LIN {X 55.431,Y 89.332,Z 63.210,A 180.000,B 0.000,C 180.000} C_DIS
LIN {X 55.354,Y 89.351,Z 63.208,A 180.000,B 0.000,C 180.000} C_DIS
LIN {X 55.279,Y 89.372,Z 63.205,A 180.000,B 0.000,C 180.000} C_DIS
LIN {X 55.127,Y 89.416,Z 63.199,A 180.000,B 0.000,C 180.000} C_DIS
LIN {X 55.052,Y 89.438,Z 63.197,A 180.000,B 0.000,C 180.000} C_DIS
LIN {X 54.901,Y 89.482,Z 63.191,A 180.000,B 0.000,C 180.000} C_DIS
LIN {X 54.749,Y 89.526,Z 63.186,A 180.000,B 0.000,C 180.000} C_DIS
LIN {X 54.674,Y 89.548,Z 63.183,A 180.000,B 0.000,C 180.000} C_DIS
LIN {X 54.599,Y 89.572,Z 63.180,A 180.000,B 0.000,C 180.000} C_DIS
LIN {X 54.524,Y 89.598,Z 63.177,A 180.000,B 0.000,C 180.000} C_DIS
LIN {X 54.450,Y 89.625,Z 63.175,A 180.000,B 0.000,C 180.000} C_DIS
LIN {X 54.302,Y 89.678,Z 63.169,A 180.000,B 0.000,C 180.000} C_DIS
LIN {X 54.006,Y 89.785,Z 63.158,A 180.000,B 0.000,C 180.000} C_DIS
LIN {X 53.932,Y 89.812,Z 63.155,A 180.000,B 0.000,C 180.000} C_DIS
LIN {X 53.858,Y 89.840,Z 63.153,A 180.000,B 0.000,C 180.000} C_DIS
LIN {X 53.786,Y 89.871,Z 63.150,A 180.000,B 0.000,C 180.000} C_DIS
LIN {X 53.352,Y 90.058,Z 63.133,A 180.000,B 0.000,C 180.000} C_DIS
LIN {X 53.280,Y 90.090,Z 63.131,A 180.000,B 0.000,C 180.000} C_DIS
LIN {X 53.208,Y 90.121,Z 63.128,A 180.000,B 0.000,C 180.000} C_DIS
LIN {X 53.136,Y 90.154,Z 63.125,A 180.000,B 0.000,C 180.000} C_DIS
LIN {X 53.066,Y 90.189,Z 63.122,A 180.000,B 0.000,C 180.000} C_DIS
LIN {X 52.925,Y 90.261,Z 63.117,A 180.000,B 0.000,C 180.000} C_DIS
LIN {X 52.575,Y 90.440,Z 63.103,A 180.000,B 0.000,C 180.000} C_DIS
LIN {X 52.504,Y 90.475,Z 63.100,A 180.000,B 0.000,C 180.000} C_DIS
LIN {X 52.435,Y 90.513,Z 63.098,A 180.000,B 0.000,C 180.000} C_DIS
LIN {X 52.367,Y 90.552,Z 63.095,A 180.000,B 0.000,C 180.000} C_DIS
LIN {X 51.892,Y 90.833,Z 63.076,A 180.000,B 0.000,C 180.000} C_DIS
LIN {X 51.825,Y 90.873,Z 63.073,A 180.000,B 0.000,C 180.000} C_DIS
LIN {X 51.758,Y 90.915,Z 63.070,A 180.000,B 0.000,C 180.000} C_DIS
LIN {X 51.692,Y 90.959,Z 63.067,A 180.000,B 0.000,C 180.000} C_DIS
LIN {X 51.302,Y 91.224,Z 63.051,A 180.000,B 0.000,C 180.000} C_DIS
LIN {X 51.236,Y 91.268,Z 63.048,A 180.000,B 0.000,C 180.000} C_DIS
LIN {X 51.171,Y 91.313,Z 63.045,A 180.000,B 0.000,C 180.000} C_DIS
LIN {X 51.107,Y 91.359,Z 63.043,A 180.000,B 0.000,C 180.000} C_DIS
LIN {X 51.045,Y 91.406,Z 63.040,A 180.000,B 0.000,C 180.000} C_DIS
LIN {X 50.609,Y 91.744,Z 63.021,A 180.000,B 0.000,C 180.000} C_DIS
LIN {X 50.547,Y 91.792,Z 63.018,A 180.000,B 0.000,C 180.000} C_DIS
LIN {X 50.486,Y 91.842,Z 63.015,A 180.000,B 0.000,C 180.000} C_DIS
LIN {X 50.426,Y 91.894,Z 63.012,A 180.000,B 0.000,C 180.000} C_DIS
LIN {X 50.013,Y 92.258,Z 62.993,A 180.000,B 0.000,C 180.000} C_DIS
LIN {X 49.954,Y 92.310,Z 62.990,A 180.000,B 0.000,C 180.000} C_DIS
LIN {X 49.896,Y 92.364,Z 62.988,A 180.000,B 0.000,C 180.000} C_DIS
LIN {X 49.840,Y 92.419,Z 62.985,A 180.000,B 0.000,C 180.000} C_DIS
LIN {X 49.450,Y 92.809,Z 62.966,A 180.000,B 0.000,C 180.000} C_DIS
LIN {X 49.394,Y 92.865,Z 62.963,A 180.000,B 0.000,C 180.000} C_DIS
LIN {X 49.340,Y 92.921,Z 62.960,A 180.000,B 0.000,C 180.000} C_DIS
LIN {X 49.287,Y 92.980,Z 62.957,A 180.000,B 0.000,C 180.000} C_DIS
LIN {X 48.975,Y 93.334,Z 62.941,A 180.000,B 0.000,C 180.000} C_DIS
LIN {X 48.923,Y 93.393,Z 62.938,A 180.000,B 0.000,C 180.000} C_DIS
LIN {X 48.871,Y 93.453,Z 62.935,A 180.000,B 0.000,C 180.000} C_DIS
LIN {X 48.820,Y 93.513,Z 62.933,A 180.000,B 0.000,C 180.000} C_DIS
LIN {X 48.771,Y 93.575,Z 62.930,A 180.000,B 0.000,C 180.000} C_DIS
LIN {X 48.433,Y 94.010,Z 62.911,A 180.000,B 0.000,C 180.000} C_DIS
LIN {X 48.385,Y 94.072,Z 62.908,A 180.000,B 0.000,C 180.000} C_DIS
LIN {X 48.338,Y 94.136,Z 62.905,A 180.000,B 0.000,C 180.000} C_DIS
LIN {X 48.293,Y 94.200,Z 62.902,A 180.000,B 0.000,C 180.000} C_DIS
LIN {X 48.204,Y 94.331,Z 62.897,A 180.000,B 0.000,C 180.000} C_DIS
LIN {X 47.983,Y 94.656,Z 62.883,A 180.000,B 0.000,C 180.000} C_DIS
LIN {X 47.939,Y 94.721,Z 62.880,A 180.000,B 0.000,C 180.000} C_DIS
LIN {X 47.896,Y 94.788,Z 62.878,A 180.000,B 0.000,C 180.000} C_DIS
LIN {X 47.855,Y 94.855,Z 62.875,A 180.000,B 0.000,C 180.000} C_DIS
LIN {X 47.615,Y 95.262,Z 62.858,A 180.000,B 0.000,C 180.000} C_DIS
LIN {X 47.575,Y 95.329,Z 62.856,A 180.000,B 0.000,C 180.000} C_DIS
LIN {X 47.535,Y 95.397,Z 62.853,A 180.000,B 0.000,C 180.000} C_DIS
LIN {X 47.496,Y 95.466,Z 62.850,A 180.000,B 0.000,C 180.000} C_DIS
LIN {X 47.459,Y 95.536,Z 62.847,A 180.000,B 0.000,C 180.000} C_DIS
LIN {X 47.388,Y 95.676,Z 62.842,A 180.000,B 0.000,C 180.000} C_DIS
LIN {X 47.209,Y 96.027,Z 62.828,A 180.000,B 0.000,C 180.000} C_DIS
LIN {X 47.173,Y 96.097,Z 62.825,A 180.000,B 0.000,C 180.000} C_DIS
LIN {X 47.139,Y 96.168,Z 62.823,A 180.000,B 0.000,C 180.000} C_DIS
LIN {X 47.107,Y 96.240,Z 62.820,A 180.000,B 0.000,C 180.000} C_DIS
LIN {X 47.044,Y 96.384,Z 62.814,A 180.000,B 0.000,C 180.000} C_DIS
LIN {X 47.013,Y 96.457,Z 62.812,A 180.000,B 0.000,C 180.000} C_DIS
LIN {X 46.951,Y 96.601,Z 62.806,A 180.000,B 0.000,C 180.000} C_DIS
LIN {X 46.888,Y 96.746,Z 62.801,A 180.000,B 0.000,C 180.000} C_DIS
LIN {X 46.857,Y 96.818,Z 62.798,A 180.000,B 0.000,C 180.000} C_DIS
LIN {X 46.827,Y 96.891,Z 62.795,A 180.000,B 0.000,C 180.000} C_DIS
LIN {X 46.800,Y 96.965,Z 62.792,A 180.000,B 0.000,C 180.000} C_DIS
LIN {X 46.773,Y 97.039,Z 62.790,A 180.000,B 0.000,C 180.000} C_DIS
LIN {X 46.720,Y 97.187,Z 62.784,A 180.000,B 0.000,C 180.000} C_DIS
LIN {X 46.639,Y 97.409,Z 62.776,A 180.000,B 0.000,C 180.000} C_DIS
LIN {X 46.613,Y 97.483,Z 62.773,A 180.000,B 0.000,C 180.000} C_DIS
LIN {X 46.586,Y 97.557,Z 62.770,A 180.000,B 0.000,C 180.000} C_DIS
LIN {X 46.561,Y 97.632,Z 62.768,A 180.000,B 0.000,C 180.000} C_DIS
LIN {X 46.538,Y 97.707,Z 62.765,A 180.000,B 0.000,C 180.000} C_DIS
LIN {X 46.494,Y 97.859,Z 62.759,A 180.000,B 0.000,C 180.000} C_DIS
LIN {X 46.472,Y 97.934,Z 62.757,A 180.000,B 0.000,C 180.000} C_DIS
LIN {X 46.428,Y 98.085,Z 62.751,A 180.000,B 0.000,C 180.000} C_DIS
LIN {X 46.384,Y 98.237,Z 62.746,A 180.000,B 0.000,C 180.000} C_DIS
LIN {X 46.362,Y 98.312,Z 62.743,A 180.000,B 0.000,C 180.000} C_DIS
LIN {X 46.342,Y 98.388,Z 62.740,A 180.000,B 0.000,C 180.000} C_DIS
LIN {X 46.324,Y 98.465,Z 62.737,A 180.000,B 0.000,C 180.000} C_DIS
LIN {X 46.307,Y 98.542,Z 62.735,A 180.000,B 0.000,C 180.000} C_DIS
LIN {X 46.272,Y 98.696,Z 62.729,A 180.000,B 0.000,C 180.000} C_DIS
LIN {X 46.221,Y 98.926,Z 62.721,A 180.000,B 0.000,C 180.000} C_DIS
LIN {X 46.204,Y 99.003,Z 62.718,A 180.000,B 0.000,C 180.000} C_DIS
LIN {X 46.186,Y 99.080,Z 62.715,A 180.000,B 0.000,C 180.000} C_DIS
LIN {X 46.171,Y 99.157,Z 62.713,A 180.000,B 0.000,C 180.000} C_DIS
LIN {X 46.157,Y 99.235,Z 62.710,A 180.000,B 0.000,C 180.000} C_DIS
LIN {X 46.133,Y 99.390,Z 62.704,A 180.000,B 0.000,C 180.000} C_DIS
LIN {X 46.120,Y 99.468,Z 62.702,A 180.000,B 0.000,C 180.000} C_DIS
LIN {X 46.096,Y 99.624,Z 62.696,A 180.000,B 0.000,C 180.000} C_DIS
LIN {X 46.071,Y 99.779,Z 62.691,A 180.000,B 0.000,C 180.000} C_DIS
LIN {X 46.059,Y 99.857,Z 62.688,A 180.000,B 0.000,C 180.000} C_DIS
LIN {X 46.048,Y 99.935,Z 62.685,A 180.000,B 0.000,C 180.000} C_DIS
LIN {X 46.040,Y 100.013,Z 62.682,A 180.000,B 0.000,C 180.000} C_DIS
LIN {X 46.025,Y 100.170,Z 62.677,A 180.000,B 0.000,C 180.000} C_DIS
LIN {X 46.010,Y 100.327,Z 62.672,A 180.000,B 0.000,C 180.000} C_DIS
LIN {X 45.995,Y 100.484,Z 62.666,A 180.000,B 0.000,C 180.000} C_DIS
LIN {X 45.988,Y 100.562,Z 62.664,A 180.000,B 0.000,C 180.000} C_DIS
LIN {X 45.980,Y 100.640,Z 62.661,A 180.000,B 0.000,C 180.000} C_DIS
LIN {X 45.974,Y 100.719,Z 62.659,A 180.000,B 0.000,C 180.000} C_DIS
LIN {X 45.971,Y 100.798,Z 62.656,A 180.000,B 0.000,C 180.000} C_DIS
LIN {X 45.968,Y 100.876,Z 62.654,A 180.000,B 0.000,C 180.000} C_DIS
LIN {X 45.966,Y 100.955,Z 62.651,A 180.000,B 0.000,C 180.000} C_DIS
LIN {X 45.963,Y 101.034,Z 62.649,A 180.000,B 0.000,C 180.000} C_DIS
LIN {X 45.958,Y 101.191,Z 62.644,A 180.000,B 0.000,C 180.000} C_DIS
LIN {X 45.954,Y 101.349,Z 62.639,A 180.000,B 0.000,C 180.000} C_DIS
LIN {X 45.950,Y 101.506,Z 62.634,A 180.000,B 0.000,C 180.000} C_DIS
LIN {X 45.954,Y 101.664,Z 62.629,A 180.000,B 0.000,C 180.000} C_DIS
LIN {X 45.959,Y 101.821,Z 62.624,A 180.000,B 0.000,C 180.000} C_DIS
LIN {X 45.964,Y 101.978,Z 62.620,A 180.000,B 0.000,C 180.000} C_DIS
LIN {X 45.969,Y 102.136,Z 62.615,A 180.000,B 0.000,C 180.000} C_DIS
LIN {X 45.975,Y 102.293,Z 62.611,A 180.000,B 0.000,C 180.000} C_DIS
LIN {X 45.989,Y 102.450,Z 62.606,A 180.000,B 0.000,C 180.000} C_DIS
LIN {X 46.004,Y 102.607,Z 62.602,A 180.000,B 0.000,C 180.000} C_DIS
LIN {X 46.018,Y 102.764,Z 62.597,A 180.000,B 0.000,C 180.000} C_DIS
LIN {X 46.033,Y 102.920,Z 62.593,A 180.000,B 0.000,C 180.000} C_DIS
LIN {X 46.049,Y 103.077,Z 62.589,A 180.000,B 0.000,C 180.000} C_DIS
LIN {X 46.073,Y 103.233,Z 62.585,A 180.000,B 0.000,C 180.000} C_DIS
LIN {X 46.098,Y 103.388,Z 62.581,A 180.000,B 0.000,C 180.000} C_DIS
LIN {X 46.122,Y 103.544,Z 62.577,A 180.000,B 0.000,C 180.000} C_DIS
LIN {X 46.147,Y 103.700,Z 62.573,A 180.000,B 0.000,C 180.000} C_DIS
LIN {X 46.173,Y 103.855,Z 62.570,A 180.000,B 0.000,C 180.000} C_DIS
LIN {X 46.206,Y 104.009,Z 62.566,A 180.000,B 0.000,C 180.000} C_DIS
LIN {X 46.241,Y 104.163,Z 62.562,A 180.000,B 0.000,C 180.000} C_DIS
LIN {X 46.275,Y 104.316,Z 62.559,A 180.000,B 0.000,C 180.000} C_DIS
LIN {X 46.309,Y 104.470,Z 62.556,A 180.000,B 0.000,C 180.000} C_DIS
LIN {X 46.345,Y 104.623,Z 62.552,A 180.000,B 0.000,C 180.000} C_DIS
LIN {X 46.388,Y 104.775,Z 62.549,A 180.000,B 0.000,C 180.000} C_DIS
LIN {X 46.432,Y 104.926,Z 62.546,A 180.000,B 0.000,C 180.000} C_DIS
LIN {X 46.476,Y 105.077,Z 62.543,A 180.000,B 0.000,C 180.000} C_DIS
LIN {X 46.520,Y 105.229,Z 62.540,A 180.000,B 0.000,C 180.000} C_DIS
LIN {X 46.565,Y 105.380,Z 62.537,A 180.000,B 0.000,C 180.000} C_DIS
LIN {X 46.617,Y 105.528,Z 62.534,A 180.000,B 0.000,C 180.000} C_DIS
LIN {X 46.670,Y 105.676,Z 62.532,A 180.000,B 0.000,C 180.000} C_DIS
LIN {X 46.724,Y 105.825,Z 62.529,A 180.000,B 0.000,C 180.000} C_DIS
LIN {X 46.777,Y 105.973,Z 62.527,A 180.000,B 0.000,C 180.000} C_DIS
LIN {X 46.893,Y 106.266,Z 62.522,A 180.000,B 0.000,C 180.000} C_DIS
LIN {X 47.018,Y 106.555,Z 62.518,A 180.000,B 0.000,C 180.000} C_DIS
LIN {X 47.144,Y 106.843,Z 62.514,A 180.000,B 0.000,C 180.000} C_DIS
LIN {X 47.286,Y 107.125,Z 62.511,A 180.000,B 0.000,C 180.000} C_DIS
LIN {X 47.429,Y 107.405,Z 62.508,A 180.000,B 0.000,C 180.000} C_DIS
LIN {X 47.581,Y 107.681,Z 62.505,A 180.000,B 0.000,C 180.000} C_DIS
LIN {X 47.741,Y 107.952,Z 62.503,A 180.000,B 0.000,C 180.000} C_DIS
LIN {X 47.903,Y 108.223,Z 62.502,A 180.000,B 0.000,C 180.000} C_DIS
LIN {X 48.079,Y 108.484,Z 62.501,A 180.000,B 0.000,C 180.000} C_DIS
LIN {X 48.256,Y 108.745,Z 62.500,A 180.000,B 0.000,C 180.000} C_DIS
LIN {X 48.390,Y 108.933,Z 62.500,A 180.000,B 0.000,C 180.000} C_DIS
; Cutting Move Starts
LIN {X 48.450,Y 109.012,Z 62.500,A 180.000,B 0.000,C 180.000} C_DIS
LIN {X 48.759,Y 109.410,Z 62.500,A 180.000,B 0.000,C 180.000} C_DIS
LIN {X 48.807,Y 109.472,Z 62.500,A 180.000,B 0.000,C 180.000} C_DIS
LIN {X 48.907,Y 109.589,Z 62.500,A 180.000,B 0.000,C 180.000} C_DIS
LIN {X 49.223,Y 109.947,Z 62.500,A 180.000,B 0.000,C 180.000} C_DIS
LIN {X 49.344,Y 110.083,Z 62.500,A 180.000,B 0.000,C 180.000} C_DIS
LIN {X 49.384,Y 110.126,Z 62.500,A 180.000,B 0.000,C 180.000} C_DIS
LIN {X 49.523,Y 110.264,Z 62.500,A 180.000,B 0.000,C 180.000} C_DIS
LIN {X 49.742,Y 110.483,Z 62.500,A 180.000,B 0.000,C 180.000} C_DIS
LIN {X 49.880,Y 110.621,Z 62.500,A 180.000,B 0.000,C 180.000} C_DIS
LIN {X 49.923,Y 110.662,Z 62.500,A 180.000,B 0.000,C 180.000} C_DIS
LIN {X 50.059,Y 110.782,Z 62.500,A 180.000,B 0.000,C 180.000} C_DIS
LIN {X 50.416,Y 111.098,Z 62.500,A 180.000,B 0.000,C 180.000} C_DIS
LIN {X 50.535,Y 111.198,Z 62.500,A 180.000,B 0.000,C 180.000} C_DIS
LIN {X 50.595,Y 111.245,Z 62.500,A 180.000,B 0.000,C 180.000} C_DIS
LIN {X 50.996,Y 111.556,Z 62.500,A 180.000,B 0.000,C 180.000} C_DIS
LIN {X 51.131,Y 111.659,Z 62.500,A 180.000,B 0.000,C 180.000} C_DIS
LIN {X 51.241,Y 111.734,Z 62.500,A 180.000,B 0.000,C 180.000} C_DIS
LIN {X 51.668,Y 112.025,Z 62.500,A 180.000,B 0.000,C 180.000} C_DIS
LIN {X 51.769,Y 112.092,Z 62.500,A 180.000,B 0.000,C 180.000} C_DIS
LIN {X 51.847,Y 112.140,Z 62.500,A 180.000,B 0.000,C 180.000} C_DIS
LIN {X 52.383,Y 112.457,Z 62.500,A 180.000,B 0.000,C 180.000} C_DIS
LIN {X 52.562,Y 112.554,Z 62.500,A 180.000,B 0.000,C 180.000} C_DIS
LIN {X 53.059,Y 112.807,Z 62.500,A 180.000,B 0.000,C 180.000} C_DIS
LIN {X 53.098,Y 112.827,Z 62.500,A 180.000,B 0.000,C 180.000} C_DIS
LIN {X 53.277,Y 112.909,Z 62.500,A 180.000,B 0.000,C 180.000} C_DIS
LIN {X 53.813,Y 113.141,Z 62.500,A 180.000,B 0.000,C 180.000} C_DIS
LIN {X 53.870,Y 113.165,Z 62.500,A 180.000,B 0.000,C 180.000} C_DIS
LIN {X 53.992,Y 113.210,Z 62.500,A 180.000,B 0.000,C 180.000} C_DIS
LIN {X 54.528,Y 113.403,Z 62.500,A 180.000,B 0.000,C 180.000} C_DIS
LIN {X 54.707,Y 113.462,Z 62.500,A 180.000,B 0.000,C 180.000} C_DIS
LIN {X 55.243,Y 113.618,Z 62.500,A 180.000,B 0.000,C 180.000} C_DIS
LIN {X 55.422,Y 113.666,Z 62.500,A 180.000,B 0.000,C 180.000} C_DIS
LIN {X 55.575,Y 113.701,Z 62.500,A 180.000,B 0.000,C 180.000} C_DIS
LIN {X 55.958,Y 113.786,Z 62.500,A 180.000,B 0.000,C 180.000} C_DIS
LIN {X 56.137,Y 113.826,Z 62.500,A 180.000,B 0.000,C 180.000} C_DIS
LIN {X 56.316,Y 113.855,Z 62.500,A 180.000,B 0.000,C 180.000} C_DIS
LIN {X 56.852,Y 113.940,Z 62.500,A 180.000,B 0.000,C 180.000} C_DIS
LIN {X 57.031,Y 113.962,Z 62.500,A 180.000,B 0.000,C 180.000} C_DIS
LIN {X 57.567,Y 114.013,Z 62.500,A 180.000,B 0.000,C 180.000} C_DIS
LIN {X 57.746,Y 114.027,Z 62.500,A 180.000,B 0.000,C 180.000} C_DIS
LIN {X 57.925,Y 114.033,Z 62.500,A 180.000,B 0.000,C 180.000} C_DIS
LIN {X 58.282,Y 114.044,Z 62.500,A 180.000,B 0.000,C 180.000} C_DIS
LIN {X 58.461,Y 114.050,Z 62.500,A 180.000,B 0.000,C 180.000} C_DIS
LIN {X 58.640,Y 114.047,Z 62.500,A 180.000,B 0.000,C 180.000} C_DIS
LIN {X 59.176,Y 114.030,Z 62.500,A 180.000,B 0.000,C 180.000} C_DIS
LIN {X 59.355,Y 114.020,Z 62.500,A 180.000,B 0.000,C 180.000} C_DIS
LIN {X 59.534,Y 114.003,Z 62.500,A 180.000,B 0.000,C 180.000} C_DIS
LIN {X 59.891,Y 113.969,Z 62.500,A 180.000,B 0.000,C 180.000} C_DIS
LIN {X 60.070,Y 113.951,Z 62.500,A 180.000,B 0.000,C 180.000} C_DIS
LIN {X 60.249,Y 113.924,Z 62.500,A 180.000,B 0.000,C 180.000} C_DIS
LIN {X 60.606,Y 113.868,Z 62.500,A 180.000,B 0.000,C 180.000} C_DIS
LIN {X 60.785,Y 113.839,Z 62.500,A 180.000,B 0.000,C 180.000} C_DIS
LIN {X 60.964,Y 113.804,Z 62.500,A 180.000,B 0.000,C 180.000} C_DIS
LIN {X 61.500,Y 113.684,Z 62.500,A 180.000,B 0.000,C 180.000} C_DIS
LIN {X 61.679,Y 113.640,Z 62.500,A 180.000,B 0.000,C 180.000} C_DIS
LIN {X 61.858,Y 113.588,Z 62.500,A 180.000,B 0.000,C 180.000} C_DIS
LIN {X 62.215,Y 113.484,Z 62.500,A 180.000,B 0.000,C 180.000} C_DIS
LIN {X 62.394,Y 113.431,Z 62.500,A 180.000,B 0.000,C 180.000} C_DIS
LIN {X 62.573,Y 113.367,Z 62.500,A 180.000,B 0.000,C 180.000} C_DIS
LIN {X 62.930,Y 113.238,Z 62.500,A 180.000,B 0.000,C 180.000} C_DIS
LIN {X 63.109,Y 113.173,Z 62.500,A 180.000,B 0.000,C 180.000} C_DIS
LIN {X 63.130,Y 113.165,Z 62.500,A 180.000,B 0.000,C 180.000} C_DIS
LIN {X 63.288,Y 113.097,Z 62.500,A 180.000,B 0.000,C 180.000} C_DIS
LIN {X 63.645,Y 112.943,Z 62.500,A 180.000,B 0.000,C 180.000} C_DIS
LIN {X 63.824,Y 112.865,Z 62.500,A 180.000,B 0.000,C 180.000} C_DIS
LIN {X 63.941,Y 112.807,Z 62.500,A 180.000,B 0.000,C 180.000} C_DIS
LIN {X 64.360,Y 112.594,Z 62.500,A 180.000,B 0.000,C 180.000} C_DIS
LIN {X 64.539,Y 112.501,Z 62.500,A 180.000,B 0.000,C 180.000} C_DIS
LIN {X 64.630,Y 112.450,Z 62.500,A 180.000,B 0.000,C 180.000} C_DIS
LIN {X 65.075,Y 112.186,Z 62.500,A 180.000,B 0.000,C 180.000} C_DIS
LIN {X 65.231,Y 112.092,Z 62.500,A 180.000,B 0.000,C 180.000} C_DIS
LIN {X 65.254,Y 112.077,Z 62.500,A 180.000,B 0.000,C 180.000} C_DIS
LIN {X 65.433,Y 111.956,Z 62.500,A 180.000,B 0.000,C 180.000} C_DIS
LIN {X 65.791,Y 111.713,Z 62.500,A 180.000,B 0.000,C 180.000} C_DIS
LIN {X 65.969,Y 111.583,Z 62.500,A 180.000,B 0.000,C 180.000} C_DIS
LIN {X 66.327,Y 111.306,Z 62.500,A 180.000,B 0.000,C 180.000} C_DIS
LIN {X 66.465,Y 111.198,Z 62.500,A 180.000,B 0.000,C 180.000} C_DIS
LIN {X 66.506,Y 111.165,Z 62.500,A 180.000,B 0.000,C 180.000} C_DIS
LIN {X 66.672,Y 111.019,Z 62.500,A 180.000,B 0.000,C 180.000} C_DIS
LIN {X 66.875,Y 110.841,Z 62.500,A 180.000,B 0.000,C 180.000} C_DIS
LIN {X 67.042,Y 110.693,Z 62.500,A 180.000,B 0.000,C 180.000} C_DIS
LIN {X 67.077,Y 110.662,Z 62.500,A 180.000,B 0.000,C 180.000} C_DIS
LIN {X 67.221,Y 110.521,Z 62.500,A 180.000,B 0.000,C 180.000} C_DIS
LIN {X 67.578,Y 110.163,Z 62.500,A 180.000,B 0.000,C 180.000} C_DIS
LIN {X 67.616,Y 110.126,Z 62.500,A 180.000,B 0.000,C 180.000} C_DIS
LIN {X 67.757,Y 109.970,Z 62.500,A 180.000,B 0.000,C 180.000} C_DIS
LIN {X 68.115,Y 109.564,Z 62.500,A 180.000,B 0.000,C 180.000} C_DIS
LIN {X 68.241,Y 109.410,Z 62.500,A 180.000,B 0.000,C 180.000} C_DIS
LIN {X 68.518,Y 109.053,Z 62.500,A 180.000,B 0.000,C 180.000} C_DIS
LIN {X 68.651,Y 108.880,Z 62.500,A 180.000,B 0.000,C 180.000} C_DIS
LIN {X 68.655,Y 108.874,Z 62.500,A 180.000,B 0.000,C 180.000} C_DIS
LIN {X 68.778,Y 108.695,Z 62.500,A 180.000,B 0.000,C 180.000} C_DIS
LIN {X 69.021,Y 108.338,Z 62.500,A 180.000,B 0.000,C 180.000} C_DIS
LIN {X 69.137,Y 108.159,Z 62.500,A 180.000,B 0.000,C 180.000} C_DIS
LIN {X 69.454,Y 107.623,Z 62.500,A 180.000,B 0.000,C 180.000} C_DIS
LIN {X 69.545,Y 107.456,Z 62.500,A 180.000,B 0.000,C 180.000} C_DIS
LIN {X 69.733,Y 107.086,Z 62.500,A 180.000,B 0.000,C 180.000} C_DIS
LIN {X 69.824,Y 106.908,Z 62.500,A 180.000,B 0.000,C 180.000} C_DIS
LIN {X 69.902,Y 106.739,Z 62.500,A 180.000,B 0.000,C 180.000} C_DIS
LIN {X 70.139,Y 106.193,Z 62.500,A 180.000,B 0.000,C 180.000} C_DIS
LIN {X 70.208,Y 106.014,Z 62.500,A 180.000,B 0.000,C 180.000} C_DIS
LIN {X 70.401,Y 105.477,Z 62.500,A 180.000,B 0.000,C 180.000} C_DIS
LIN {X 70.439,Y 105.369,Z 62.500,A 180.000,B 0.000,C 180.000} C_DIS
LIN {X 70.460,Y 105.299,Z 62.500,A 180.000,B 0.000,C 180.000} C_DIS
LIN {X 70.617,Y 104.758,Z 62.500,A 180.000,B 0.000,C 180.000} C_DIS
LIN {X 70.665,Y 104.584,Z 62.500,A 180.000,B 0.000,C 180.000} C_DIS
LIN {X 70.705,Y 104.405,Z 62.500,A 180.000,B 0.000,C 180.000} C_DIS
LIN {X 70.796,Y 103.999,Z 62.500,A 180.000,B 0.000,C 180.000} C_DIS
LIN {X 70.824,Y 103.869,Z 62.500,A 180.000,B 0.000,C 180.000} C_DIS
LIN {X 70.855,Y 103.690,Z 62.500,A 180.000,B 0.000,C 180.000} C_DIS
LIN {X 70.940,Y 103.153,Z 62.500,A 180.000,B 0.000,C 180.000} C_DIS
LIN {X 70.962,Y 102.975,Z 62.500,A 180.000,B 0.000,C 180.000} C_DIS
LIN {X 71.012,Y 102.438,Z 62.500,A 180.000,B 0.000,C 180.000} C_DIS
LIN {X 71.027,Y 102.260,Z 62.500,A 180.000,B 0.000,C 180.000} C_DIS
LIN {X 71.033,Y 102.081,Z 62.500,A 180.000,B 0.000,C 180.000} C_DIS
LIN {X 71.044,Y 101.723,Z 62.500,A 180.000,B 0.000,C 180.000} C_DIS
LIN {X 71.050,Y 101.545,Z 62.500,A 180.000,B 0.000,C 180.000} C_DIS
LIN {X 71.047,Y 101.366,Z 62.500,A 180.000,B 0.000,C 180.000} C_DIS
LIN {X 71.030,Y 100.829,Z 62.500,A 180.000,B 0.000,C 180.000} C_DIS
LIN {X 71.021,Y 100.651,Z 62.500,A 180.000,B 0.000,C 180.000} C_DIS
LIN {X 71.004,Y 100.472,Z 62.500,A 180.000,B 0.000,C 180.000} C_DIS
LIN {X 70.970,Y 100.114,Z 62.500,A 180.000,B 0.000,C 180.000} C_DIS
LIN {X 70.952,Y 99.936,Z 62.500,A 180.000,B 0.000,C 180.000} C_DIS
LIN {X 70.925,Y 99.757,Z 62.500,A 180.000,B 0.000,C 180.000} C_DIS
LIN {X 70.840,Y 99.221,Z 62.500,A 180.000,B 0.000,C 180.000} C_DIS
LIN {X 70.805,Y 99.042,Z 62.500,A 180.000,B 0.000,C 180.000} C_DIS
LIN {X 70.718,Y 98.654,Z 62.500,A 180.000,B 0.000,C 180.000} C_DIS
LIN {X 70.685,Y 98.505,Z 62.500,A 180.000,B 0.000,C 180.000} C_DIS
LIN {X 70.642,Y 98.327,Z 62.500,A 180.000,B 0.000,C 180.000} C_DIS
LIN {X 70.617,Y 98.242,Z 62.500,A 180.000,B 0.000,C 180.000} C_DIS
LIN {X 70.486,Y 97.790,Z 62.500,A 180.000,B 0.000,C 180.000} C_DIS
LIN {X 70.439,Y 97.631,Z 62.500,A 180.000,B 0.000,C 180.000} C_DIS
LIN {X 70.432,Y 97.612,Z 62.500,A 180.000,B 0.000,C 180.000} C_DIS
LIN {X 70.369,Y 97.433,Z 62.500,A 180.000,B 0.000,C 180.000} C_DIS
LIN {X 70.240,Y 97.075,Z 62.500,A 180.000,B 0.000,C 180.000} C_DIS
LIN {X 70.175,Y 96.897,Z 62.500,A 180.000,B 0.000,C 180.000} C_DIS
LIN {X 70.100,Y 96.718,Z 62.500,A 180.000,B 0.000,C 180.000} C_DIS
LIN {X 69.902,Y 96.261,Z 62.500,A 180.000,B 0.000,C 180.000} C_DIS
LIN {X 69.867,Y 96.181,Z 62.500,A 180.000,B 0.000,C 180.000} C_DIS
LIN {X 69.779,Y 96.003,Z 62.500,A 180.000,B 0.000,C 180.000} C_DIS
LIN {X 69.545,Y 95.544,Z 62.500,A 180.000,B 0.000,C 180.000} C_DIS
LIN {X 69.504,Y 95.466,Z 62.500,A 180.000,B 0.000,C 180.000} C_DIS
LIN {X 69.401,Y 95.288,Z 62.500,A 180.000,B 0.000,C 180.000} C_DIS
LIN {X 69.187,Y 94.927,Z 62.500,A 180.000,B 0.000,C 180.000} C_DIS
LIN {X 69.081,Y 94.751,Z 62.500,A 180.000,B 0.000,C 180.000} C_DIS
LIN {X 69.008,Y 94.644,Z 62.500,A 180.000,B 0.000,C 180.000} C_DIS
LIN {X 68.717,Y 94.215,Z 62.500,A 180.000,B 0.000,C 180.000} C_DIS
LIN {X 68.651,Y 94.120,Z 62.500,A 180.000,B 0.000,C 180.000} C_DIS
LIN {X 68.587,Y 94.036,Z 62.500,A 180.000,B 0.000,C 180.000} C_DIS
LIN {X 68.293,Y 93.657,Z 62.500,A 180.000,B 0.000,C 180.000} C_DIS
LIN {X 68.170,Y 93.500,Z 62.500,A 180.000,B 0.000,C 180.000} C_DIS
LIN {X 68.115,Y 93.436,Z 62.500,A 180.000,B 0.000,C 180.000} C_DIS
LIN {X 67.698,Y 92.964,Z 62.500,A 180.000,B 0.000,C 180.000} C_DIS
LIN {X 67.578,Y 92.837,Z 62.500,A 180.000,B 0.000,C 180.000} C_DIS
LIN {X 67.169,Y 92.427,Z 62.500,A 180.000,B 0.000,C 180.000} C_DIS
LIN {X 67.061,Y 92.325,Z 62.500,A 180.000,B 0.000,C 180.000} C_DIS
LIN {X 67.042,Y 92.307,Z 62.500,A 180.000,B 0.000,C 180.000} C_DIS
LIN {X 66.976,Y 92.249,Z 62.500,A 180.000,B 0.000,C 180.000} C_DIS
LIN {X 66.571,Y 91.891,Z 62.500,A 180.000,B 0.000,C 180.000} C_DIS
LIN {X 66.506,Y 91.835,Z 62.500,A 180.000,B 0.000,C 180.000} C_DIS
LIN {X 66.350,Y 91.712,Z 62.500,A 180.000,B 0.000,C 180.000} C_DIS
LIN {X 65.969,Y 91.417,Z 62.500,A 180.000,B 0.000,C 180.000} C_DIS
LIN {X 65.887,Y 91.355,Z 62.500,A 180.000,B 0.000,C 180.000} C_DIS
LIN {X 65.791,Y 91.287,Z 62.500,A 180.000,B 0.000,C 180.000} C_DIS
LIN {X 65.364,Y 90.997,Z 62.500,A 180.000,B 0.000,C 180.000} C_DIS
LIN {X 65.254,Y 90.923,Z 62.500,A 180.000,B 0.000,C 180.000} C_DIS
LIN {X 65.083,Y 90.818,Z 62.500,A 180.000,B 0.000,C 180.000} C_DIS
LIN {X 64.718,Y 90.603,Z 62.500,A 180.000,B 0.000,C 180.000} C_DIS
LIN {X 64.539,Y 90.499,Z 62.500,A 180.000,B 0.000,C 180.000} C_DIS
LIN {X 64.467,Y 90.461,Z 62.500,A 180.000,B 0.000,C 180.000} C_DIS
LIN {X 64.003,Y 90.224,Z 62.500,A 180.000,B 0.000,C 180.000} C_DIS
LIN {X 63.824,Y 90.135,Z 62.500,A 180.000,B 0.000,C 180.000} C_DIS
LIN {X 63.752,Y 90.103,Z 62.500,A 180.000,B 0.000,C 180.000} C_DIS
LIN {X 63.288,Y 89.903,Z 62.500,A 180.000,B 0.000,C 180.000} C_DIS
LIN {X 63.109,Y 89.827,Z 62.500,A 180.000,B 0.000,C 180.000} C_DIS
LIN {X 62.930,Y 89.762,Z 62.500,A 180.000,B 0.000,C 180.000} C_DIS
LIN {X 62.573,Y 89.633,Z 62.500,A 180.000,B 0.000,C 180.000} C_DIS
LIN {X 62.394,Y 89.569,Z 62.500,A 180.000,B 0.000,C 180.000} C_DIS
LIN {X 62.387,Y 89.567,Z 62.500,A 180.000,B 0.000,C 180.000} C_DIS
LIN {X 62.215,Y 89.516,Z 62.500,A 180.000,B 0.000,C 180.000} C_DIS
LIN {X 61.777,Y 89.388,Z 62.500,A 180.000,B 0.000,C 180.000} C_DIS
LIN {X 61.679,Y 89.360,Z 62.500,A 180.000,B 0.000,C 180.000} C_DIS
LIN {X 61.500,Y 89.316,Z 62.500,A 180.000,B 0.000,C 180.000} C_DIS
LIN {X 60.964,Y 89.196,Z 62.500,A 180.000,B 0.000,C 180.000} C_DIS
LIN {X 60.785,Y 89.161,Z 62.500,A 180.000,B 0.000,C 180.000} C_DIS
LIN {X 60.606,Y 89.132,Z 62.500,A 180.000,B 0.000,C 180.000} C_DIS
LIN {X 60.249,Y 89.076,Z 62.500,A 180.000,B 0.000,C 180.000} C_DIS
LIN {X 60.070,Y 89.049,Z 62.500,A 180.000,B 0.000,C 180.000} C_DIS
LIN {X 59.892,Y 89.031,Z 62.500,A 180.000,B 0.000,C 180.000} C_DIS
LIN {X 59.534,Y 88.997,Z 62.500,A 180.000,B 0.000,C 180.000} C_DIS
LIN {X 59.355,Y 88.980,Z 62.500,A 180.000,B 0.000,C 180.000} C_DIS
LIN {X 59.176,Y 88.970,Z 62.500,A 180.000,B 0.000,C 180.000} C_DIS
LIN {X 58.640,Y 88.953,Z 62.500,A 180.000,B 0.000,C 180.000} C_DIS
LIN {X 58.461,Y 88.950,Z 62.500,A 180.000,B 0.000,C 180.000} C_DIS
LIN {X 58.282,Y 88.956,Z 62.500,A 180.000,B 0.000,C 180.000} C_DIS
LIN {X 57.925,Y 88.967,Z 62.500,A 180.000,B 0.000,C 180.000} C_DIS
LIN {X 57.746,Y 88.973,Z 62.500,A 180.000,B 0.000,C 180.000} C_DIS
LIN {X 57.567,Y 88.987,Z 62.500,A 180.000,B 0.000,C 180.000} C_DIS
LIN {X 57.031,Y 89.038,Z 62.500,A 180.000,B 0.000,C 180.000} C_DIS
LIN {X 56.852,Y 89.060,Z 62.500,A 180.000,B 0.000,C 180.000} C_DIS
LIN {X 56.316,Y 89.145,Z 62.500,A 180.000,B 0.000,C 180.000} C_DIS
LIN {X 56.137,Y 89.174,Z 62.500,A 180.000,B 0.000,C 180.000} C_DIS
LIN {X 55.977,Y 89.209,Z 62.500,A 180.000,B 0.000,C 180.000} C_DIS
LIN {X 55.601,Y 89.293,Z 62.500,A 180.000,B 0.000,C 180.000} C_DIS
LIN {X 55.422,Y 89.334,Z 62.500,A 180.000,B 0.000,C 180.000} C_DIS
LIN {X 55.243,Y 89.382,Z 62.500,A 180.000,B 0.000,C 180.000} C_DIS
LIN {X 54.707,Y 89.538,Z 62.500,A 180.000,B 0.000,C 180.000} C_DIS
LIN {X 54.613,Y 89.567,Z 62.500,A 180.000,B 0.000,C 180.000} C_DIS
LIN {X 54.528,Y 89.597,Z 62.500,A 180.000,B 0.000,C 180.000} C_DIS
LIN {X 53.992,Y 89.790,Z 62.500,A 180.000,B 0.000,C 180.000} C_DIS
LIN {X 53.813,Y 89.859,Z 62.500,A 180.000,B 0.000,C 180.000} C_DIS
LIN {X 53.455,Y 90.014,Z 62.500,A 180.000,B 0.000,C 180.000} C_DIS
LIN {X 53.248,Y 90.103,Z 62.500,A 180.000,B 0.000,C 180.000} C_DIS
LIN {X 53.098,Y 90.173,Z 62.500,A 180.000,B 0.000,C 180.000} C_DIS
LIN {X 52.919,Y 90.264,Z 62.500,A 180.000,B 0.000,C 180.000} C_DIS
LIN {X 52.533,Y 90.461,Z 62.500,A 180.000,B 0.000,C 180.000} C_DIS
LIN {X 52.383,Y 90.543,Z 62.500,A 180.000,B 0.000,C 180.000} C_DIS
LIN {X 51.847,Y 90.860,Z 62.500,A 180.000,B 0.000,C 180.000} C_DIS
LIN {X 51.668,Y 90.975,Z 62.500,A 180.000,B 0.000,C 180.000} C_DIS
LIN {X 51.310,Y 91.218,Z 62.500,A 180.000,B 0.000,C 180.000} C_DIS
LIN {X 51.131,Y 91.341,Z 62.500,A 180.000,B 0.000,C 180.000} C_DIS
LIN {X 51.113,Y 91.355,Z 62.500,A 180.000,B 0.000,C 180.000} C_DIS
LIN {X 50.953,Y 91.478,Z 62.500,A 180.000,B 0.000,C 180.000} C_DIS
LIN {X 50.595,Y 91.755,Z 62.500,A 180.000,B 0.000,C 180.000} C_DIS
LIN {X 50.429,Y 91.891,Z 62.500,A 180.000,B 0.000,C 180.000} C_DIS
LIN {X 50.024,Y 92.249,Z 62.500,A 180.000,B 0.000,C 180.000} C_DIS
LIN {X 49.880,Y 92.379,Z 62.500,A 180.000,B 0.000,C 180.000} C_DIS
LIN {X 49.831,Y 92.427,Z 62.500,A 180.000,B 0.000,C 180.000} C_DIS
LIN {X 49.474,Y 92.785,Z 62.500,A 180.000,B 0.000,C 180.000} C_DIS
LIN {X 49.344,Y 92.917,Z 62.500,A 180.000,B 0.000,C 180.000} C_DIS
LIN {X 49.302,Y 92.964,Z 62.500,A 180.000,B 0.000,C 180.000} C_DIS
LIN {X 48.986,Y 93.321,Z 62.500,A 180.000,B 0.000,C 180.000} C_DIS
LIN {X 48.830,Y 93.500,Z 62.500,A 180.000,B 0.000,C 180.000} C_DIS
LIN {X 48.807,Y 93.528,Z 62.500,A 180.000,B 0.000,C 180.000} C_DIS
LIN {X 48.690,Y 93.679,Z 62.500,A 180.000,B 0.000,C 180.000} C_DIS
LIN {X 48.413,Y 94.036,Z 62.500,A 180.000,B 0.000,C 180.000} C_DIS
LIN {X 48.283,Y 94.215,Z 62.500,A 180.000,B 0.000,C 180.000} C_DIS
LIN {X 48.040,Y 94.573,Z 62.500,A 180.000,B 0.000,C 180.000} C_DIS
LIN {X 47.919,Y 94.751,Z 62.500,A 180.000,B 0.000,C 180.000} C_DIS
LIN {X 47.914,Y 94.760,Z 62.500,A 180.000,B 0.000,C 180.000} C_DIS
LIN {X 47.811,Y 94.930,Z 62.500,A 180.000,B 0.000,C 180.000} C_DIS
LIN {X 47.556,Y 95.361,Z 62.500,A 180.000,B 0.000,C 180.000} C_DIS
LIN {X 47.496,Y 95.466,Z 62.500,A 180.000,B 0.000,C 180.000} C_DIS
LIN {X 47.404,Y 95.645,Z 62.500,A 180.000,B 0.000,C 180.000} C_DIS
LIN {X 47.198,Y 96.048,Z 62.500,A 180.000,B 0.000,C 180.000} C_DIS
LIN {X 47.133,Y 96.181,Z 62.500,A 180.000,B 0.000,C 180.000} C_DIS
LIN {X 47.055,Y 96.360,Z 62.500,A 180.000,B 0.000,C 180.000} C_DIS
LIN {X 46.900,Y 96.718,Z 62.500,A 180.000,B 0.000,C 180.000} C_DIS
LIN {X 46.841,Y 96.856,Z 62.500,A 180.000,B 0.000,C 180.000} C_DIS
LIN {X 46.825,Y 96.897,Z 62.500,A 180.000,B 0.000,C 180.000} C_DIS
LIN {X 46.760,Y 97.075,Z 62.500,A 180.000,B 0.000,C 180.000} C_DIS
LIN {X 46.631,Y 97.433,Z 62.500,A 180.000,B 0.000,C 180.000} C_DIS
LIN {X 46.568,Y 97.612,Z 62.500,A 180.000,B 0.000,C 180.000} C_DIS
LIN {X 46.514,Y 97.790,Z 62.500,A 180.000,B 0.000,C 180.000} C_DIS
LIN {X 46.410,Y 98.148,Z 62.500,A 180.000,B 0.000,C 180.000} C_DIS
LIN {X 46.358,Y 98.327,Z 62.500,A 180.000,B 0.000,C 180.000} C_DIS
LIN {X 46.315,Y 98.505,Z 62.500,A 180.000,B 0.000,C 180.000} C_DIS
LIN {X 46.195,Y 99.042,Z 62.500,A 180.000,B 0.000,C 180.000} C_DIS
LIN {X 46.160,Y 99.221,Z 62.500,A 180.000,B 0.000,C 180.000} C_DIS
LIN {X 46.126,Y 99.434,Z 62.500,A 180.000,B 0.000,C 180.000} C_DIS
LIN {X 46.075,Y 99.757,Z 62.500,A 180.000,B 0.000,C 180.000} C_DIS
LIN {X 46.048,Y 99.936,Z 62.500,A 180.000,B 0.000,C 180.000} C_DIS
LIN {X 46.030,Y 100.114,Z 62.500,A 180.000,B 0.000,C 180.000} C_DIS
LIN {X 45.996,Y 100.472,Z 62.500,A 180.000,B 0.000,C 180.000} C_DIS
LIN {X 45.979,Y 100.651,Z 62.500,A 180.000,B 0.000,C 180.000} C_DIS
LIN {X 45.970,Y 100.829,Z 62.500,A 180.000,B 0.000,C 180.000} C_DIS
LIN {X 45.953,Y 101.366,Z 62.500,A 180.000,B 0.000,C 180.000} C_DIS
LIN {X 45.950,Y 101.545,Z 62.500,A 180.000,B 0.000,C 180.000} C_DIS
LIN {X 45.956,Y 101.723,Z 62.500,A 180.000,B 0.000,C 180.000} C_DIS
LIN {X 45.967,Y 102.081,Z 62.500,A 180.000,B 0.000,C 180.000} C_DIS
LIN {X 45.973,Y 102.260,Z 62.500,A 180.000,B 0.000,C 180.000} C_DIS
LIN {X 45.988,Y 102.438,Z 62.500,A 180.000,B 0.000,C 180.000} C_DIS
LIN {X 46.038,Y 102.975,Z 62.500,A 180.000,B 0.000,C 180.000} C_DIS
LIN {X 46.060,Y 103.153,Z 62.500,A 180.000,B 0.000,C 180.000} C_DIS
LIN {X 46.145,Y 103.690,Z 62.500,A 180.000,B 0.000,C 180.000} C_DIS
LIN {X 46.176,Y 103.869,Z 62.500,A 180.000,B 0.000,C 180.000} C_DIS
LIN {X 46.215,Y 104.047,Z 62.500,A 180.000,B 0.000,C 180.000} C_DIS
LIN {X 46.305,Y 104.449,Z 62.500,A 180.000,B 0.000,C 180.000} C_DIS
LIN {X 46.335,Y 104.584,Z 62.500,A 180.000,B 0.000,C 180.000} C_DIS
LIN {X 46.384,Y 104.762,Z 62.500,A 180.000,B 0.000,C 180.000} C_DIS
LIN {X 46.540,Y 105.299,Z 62.500,A 180.000,B 0.000,C 180.000} C_DIS
LIN {X 46.599,Y 105.477,Z 62.500,A 180.000,B 0.000,C 180.000} C_DIS
LIN {X 46.792,Y 106.014,Z 62.500,A 180.000,B 0.000,C 180.000} C_DIS
LIN {X 46.841,Y 106.144,Z 62.500,A 180.000,B 0.000,C 180.000} C_DIS
LIN {X 46.861,Y 106.193,Z 62.500,A 180.000,B 0.000,C 180.000} C_DIS
LIN {X 47.093,Y 106.729,Z 62.500,A 180.000,B 0.000,C 180.000} C_DIS
LIN {X 47.176,Y 106.908,Z 62.500,A 180.000,B 0.000,C 180.000} C_DIS
LIN {X 47.198,Y 106.952,Z 62.500,A 180.000,B 0.000,C 180.000} C_DIS
LIN {X 47.449,Y 107.444,Z 62.500,A 180.000,B 0.000,C 180.000} C_DIS
LIN {X 47.546,Y 107.623,Z 62.500,A 180.000,B 0.000,C 180.000} C_DIS
LIN {X 47.863,Y 108.159,Z 62.500,A 180.000,B 0.000,C 180.000} C_DIS
LIN {X 47.914,Y 108.240,Z 62.500,A 180.000,B 0.000,C 180.000} C_DIS
LIN {X 47.979,Y 108.338,Z 62.500,A 180.000,B 0.000,C 180.000} C_DIS
LIN {X 48.271,Y 108.767,Z 62.500,A 180.000,B 0.000,C 180.000} C_DIS
LIN {X 48.345,Y 108.874,Z 62.500,A 180.000,B 0.000,C 180.000} C_DIS
LIN {X 48.390,Y 108.933,Z 62.500,A 180.000,B 0.000,C 180.000} C_DIS
; Link Move Starts
LIN {X 48.583,Y 109.183,Z 62.500,A 180.000,B 0.000,C 180.000} C_DIS
LIN {X 48.776,Y 109.431,Z 62.498,A 180.000,B 0.000,C 180.000} C_DIS
LIN {X 48.980,Y 109.671,Z 62.496,A 180.000,B 0.000,C 180.000} C_DIS
LIN {X 49.188,Y 109.908,Z 62.492,A 180.000,B 0.000,C 180.000} C_DIS
LIN {X 49.400,Y 110.141,Z 62.488,A 180.000,B 0.000,C 180.000} C_DIS
LIN {X 49.622,Y 110.364,Z 62.483,A 180.000,B 0.000,C 180.000} C_DIS
LIN {X 49.734,Y 110.475,Z 62.481,A 180.000,B 0.000,C 180.000} C_DIS
LIN {X 49.845,Y 110.586,Z 62.478,A 180.000,B 0.000,C 180.000} C_DIS
LIN {X 49.959,Y 110.695,Z 62.475,A 180.000,B 0.000,C 180.000} C_DIS
LIN {X 50.078,Y 110.799,Z 62.471,A 180.000,B 0.000,C 180.000} C_DIS
LIN {X 50.196,Y 110.903,Z 62.468,A 180.000,B 0.000,C 180.000} C_DIS
LIN {X 50.314,Y 111.007,Z 62.464,A 180.000,B 0.000,C 180.000} C_DIS
LIN {X 50.432,Y 111.111,Z 62.460,A 180.000,B 0.000,C 180.000} C_DIS
LIN {X 50.553,Y 111.212,Z 62.456,A 180.000,B 0.000,C 180.000} C_DIS
LIN {X 50.677,Y 111.309,Z 62.452,A 180.000,B 0.000,C 180.000} C_DIS
LIN {X 50.802,Y 111.405,Z 62.448,A 180.000,B 0.000,C 180.000} C_DIS
LIN {X 50.926,Y 111.502,Z 62.444,A 180.000,B 0.000,C 180.000} C_DIS
LIN {X 51.051,Y 111.598,Z 62.439,A 180.000,B 0.000,C 180.000} C_DIS
LIN {X 51.178,Y 111.692,Z 62.434,A 180.000,B 0.000,C 180.000} C_DIS
LIN {X 51.308,Y 111.780,Z 62.429,A 180.000,B 0.000,C 180.000} C_DIS
LIN {X 51.438,Y 111.869,Z 62.424,A 180.000,B 0.000,C 180.000} C_DIS
LIN {X 51.503,Y 111.913,Z 62.422,A 180.000,B 0.000,C 180.000} C_DIS
LIN {X 51.568,Y 111.957,Z 62.419,A 180.000,B 0.000,C 180.000} C_DIS
LIN {X 51.634,Y 112.001,Z 62.417,A 180.000,B 0.000,C 180.000} C_DIS
LIN {X 51.699,Y 112.046,Z 62.414,A 180.000,B 0.000,C 180.000} C_DIS
LIN {X 51.764,Y 112.089,Z 62.411,A 180.000,B 0.000,C 180.000} C_DIS
LIN {X 51.831,Y 112.131,Z 62.409,A 180.000,B 0.000,C 180.000} C_DIS
LIN {X 51.899,Y 112.171,Z 62.406,A 180.000,B 0.000,C 180.000} C_DIS
LIN {X 51.967,Y 112.211,Z 62.403,A 180.000,B 0.000,C 180.000} C_DIS
LIN {X 52.035,Y 112.251,Z 62.401,A 180.000,B 0.000,C 180.000} C_DIS
LIN {X 52.102,Y 112.291,Z 62.398,A 180.000,B 0.000,C 180.000} C_DIS
LIN {X 52.170,Y 112.331,Z 62.395,A 180.000,B 0.000,C 180.000} C_DIS
LIN {X 52.238,Y 112.371,Z 62.392,A 180.000,B 0.000,C 180.000} C_DIS
LIN {X 52.306,Y 112.411,Z 62.389,A 180.000,B 0.000,C 180.000} C_DIS
LIN {X 52.373,Y 112.451,Z 62.387,A 180.000,B 0.000,C 180.000} C_DIS
LIN {X 52.442,Y 112.491,Z 62.384,A 180.000,B 0.000,C 180.000} C_DIS
LIN {X 52.511,Y 112.528,Z 62.381,A 180.000,B 0.000,C 180.000} C_DIS
LIN {X 52.581,Y 112.564,Z 62.378,A 180.000,B 0.000,C 180.000} C_DIS
LIN {X 52.651,Y 112.600,Z 62.376,A 180.000,B 0.000,C 180.000} C_DIS
LIN {X 52.722,Y 112.635,Z 62.373,A 180.000,B 0.000,C 180.000} C_DIS
LIN {X 52.792,Y 112.671,Z 62.370,A 180.000,B 0.000,C 180.000} C_DIS
LIN {X 52.862,Y 112.707,Z 62.367,A 180.000,B 0.000,C 180.000} C_DIS
LIN {X 52.932,Y 112.743,Z 62.365,A 180.000,B 0.000,C 180.000} C_DIS
LIN {X 53.002,Y 112.778,Z 62.362,A 180.000,B 0.000,C 180.000} C_DIS
LIN {X 53.072,Y 112.814,Z 62.359,A 180.000,B 0.000,C 180.000} C_DIS
LIN {X 53.143,Y 112.849,Z 62.356,A 180.000,B 0.000,C 180.000} C_DIS
LIN {X 53.215,Y 112.882,Z 62.354,A 180.000,B 0.000,C 180.000} C_DIS
LIN {X 53.287,Y 112.913,Z 62.351,A 180.000,B 0.000,C 180.000} C_DIS
LIN {X 53.431,Y 112.976,Z 62.345,A 180.000,B 0.000,C 180.000} C_DIS
LIN {X 53.504,Y 113.007,Z 62.343,A 180.000,B 0.000,C 180.000} C_DIS
LIN {X 53.648,Y 113.070,Z 62.337,A 180.000,B 0.000,C 180.000} C_DIS
LIN {X 53.793,Y 113.132,Z 62.332,A 180.000,B 0.000,C 180.000} C_DIS
LIN {X 53.865,Y 113.163,Z 62.329,A 180.000,B 0.000,C 180.000} C_DIS
LIN {X 53.939,Y 113.191,Z 62.326,A 180.000,B 0.000,C 180.000} C_DIS
LIN {X 54.013,Y 113.218,Z 62.323,A 180.000,B 0.000,C 180.000} C_DIS
LIN {X 54.087,Y 113.245,Z 62.321,A 180.000,B 0.000,C 180.000} C_DIS
LIN {X 54.235,Y 113.298,Z 62.315,A 180.000,B 0.000,C 180.000} C_DIS
LIN {X 54.532,Y 113.405,Z 62.304,A 180.000,B 0.000,C 180.000} C_DIS
LIN {X 54.606,Y 113.431,Z 62.301,A 180.000,B 0.000,C 180.000} C_DIS
LIN {X 54.681,Y 113.454,Z 62.299,A 180.000,B 0.000,C 180.000} C_DIS
LIN {X 54.757,Y 113.476,Z 62.296,A 180.000,B 0.000,C 180.000} C_DIS
LIN {X 55.135,Y 113.586,Z 62.282,A 180.000,B 0.000,C 180.000} C_DIS
LIN {X 55.286,Y 113.630,Z 62.277,A 180.000,B 0.000,C 180.000} C_DIS
LIN {X 55.362,Y 113.651,Z 62.274,A 180.000,B 0.000,C 180.000} C_DIS
LIN {X 55.438,Y 113.670,Z 62.271,A 180.000,B 0.000,C 180.000} C_DIS
LIN {X 55.515,Y 113.687,Z 62.268,A 180.000,B 0.000,C 180.000} C_DIS
LIN {X 55.899,Y 113.773,Z 62.255,A 180.000,B 0.000,C 180.000} C_DIS
LIN {X 56.053,Y 113.808,Z 62.249,A 180.000,B 0.000,C 180.000} C_DIS
LIN {X 56.130,Y 113.824,Z 62.246,A 180.000,B 0.000,C 180.000} C_DIS
LIN {X 56.208,Y 113.838,Z 62.244,A 180.000,B 0.000,C 180.000} C_DIS
LIN {X 56.285,Y 113.851,Z 62.241,A 180.000,B 0.000,C 180.000} C_DIS
LIN {X 56.830,Y 113.937,Z 62.222,A 180.000,B 0.000,C 180.000} C_DIS
LIN {X 56.908,Y 113.949,Z 62.219,A 180.000,B 0.000,C 180.000} C_DIS
LIN {X 56.986,Y 113.958,Z 62.216,A 180.000,B 0.000,C 180.000} C_DIS
LIN {X 57.064,Y 113.965,Z 62.213,A 180.000,B 0.000,C 180.000} C_DIS
LIN {X 57.221,Y 113.980,Z 62.208,A 180.000,B 0.000,C 180.000} C_DIS
LIN {X 57.378,Y 113.995,Z 62.202,A 180.000,B 0.000,C 180.000} C_DIS
LIN {X 57.456,Y 114.002,Z 62.200,A 180.000,B 0.000,C 180.000} C_DIS
LIN {X 57.613,Y 114.017,Z 62.194,A 180.000,B 0.000,C 180.000} C_DIS
LIN {X 57.692,Y 114.024,Z 62.191,A 180.000,B 0.000,C 180.000} C_DIS
LIN {X 57.770,Y 114.028,Z 62.189,A 180.000,B 0.000,C 180.000} C_DIS
LIN {X 57.849,Y 114.031,Z 62.186,A 180.000,B 0.000,C 180.000} C_DIS
LIN {X 58.006,Y 114.036,Z 62.180,A 180.000,B 0.000,C 180.000} C_DIS
LIN {X 58.085,Y 114.038,Z 62.178,A 180.000,B 0.000,C 180.000} C_DIS
LIN {X 58.243,Y 114.043,Z 62.172,A 180.000,B 0.000,C 180.000} C_DIS
LIN {X 58.400,Y 114.048,Z 62.167,A 180.000,B 0.000,C 180.000} C_DIS
LIN {X 58.479,Y 114.050,Z 62.164,A 180.000,B 0.000,C 180.000} C_DIS
LIN {X 58.557,Y 114.049,Z 62.161,A 180.000,B 0.000,C 180.000} C_DIS
LIN {X 58.636,Y 114.047,Z 62.158,A 180.000,B 0.000,C 180.000} C_DIS
LIN {X 58.715,Y 114.044,Z 62.156,A 180.000,B 0.000,C 180.000} C_DIS
LIN {X 58.872,Y 114.040,Z 62.150,A 180.000,B 0.000,C 180.000} C_DIS
LIN {X 59.030,Y 114.035,Z 62.145,A 180.000,B 0.000,C 180.000} C_DIS
LIN {X 59.187,Y 114.030,Z 62.139,A 180.000,B 0.000,C 180.000} C_DIS
LIN {X 59.266,Y 114.027,Z 62.136,A 180.000,B 0.000,C 180.000} C_DIS
LIN {X 59.344,Y 114.021,Z 62.134,A 180.000,B 0.000,C 180.000} C_DIS
LIN {X 59.423,Y 114.014,Z 62.131,A 180.000,B 0.000,C 180.000} C_DIS
LIN {X 59.501,Y 114.006,Z 62.128,A 180.000,B 0.000,C 180.000} C_DIS
LIN {X 59.580,Y 113.999,Z 62.125,A 180.000,B 0.000,C 180.000} C_DIS
LIN {X 59.658,Y 113.992,Z 62.123,A 180.000,B 0.000,C 180.000} C_DIS
LIN {X 59.736,Y 113.984,Z 62.120,A 180.000,B 0.000,C 180.000} C_DIS
LIN {X 59.815,Y 113.977,Z 62.117,A 180.000,B 0.000,C 180.000} C_DIS
LIN {X 59.893,Y 113.969,Z 62.114,A 180.000,B 0.000,C 180.000} C_DIS
LIN {X 59.972,Y 113.962,Z 62.112,A 180.000,B 0.000,C 180.000} C_DIS
LIN {X 60.050,Y 113.954,Z 62.109,A 180.000,B 0.000,C 180.000} C_DIS
LIN {X 60.128,Y 113.943,Z 62.106,A 180.000,B 0.000,C 180.000} C_DIS
LIN {X 60.206,Y 113.931,Z 62.103,A 180.000,B 0.000,C 180.000} C_DIS
LIN {X 60.284,Y 113.919,Z 62.101,A 180.000,B 0.000,C 180.000} C_DIS
LIN {X 60.361,Y 113.907,Z 62.098,A 180.000,B 0.000,C 180.000} C_DIS
LIN {X 60.439,Y 113.894,Z 62.095,A 180.000,B 0.000,C 180.000} C_DIS
LIN {X 60.517,Y 113.882,Z 62.092,A 180.000,B 0.000,C 180.000} C_DIS
LIN {X 60.595,Y 113.870,Z 62.090,A 180.000,B 0.000,C 180.000} C_DIS
LIN {X 60.672,Y 113.857,Z 62.087,A 180.000,B 0.000,C 180.000} C_DIS
LIN {X 60.750,Y 113.845,Z 62.084,A 180.000,B 0.000,C 180.000} C_DIS
LIN {X 60.828,Y 113.832,Z 62.082,A 180.000,B 0.000,C 180.000} C_DIS
LIN {X 60.905,Y 113.817,Z 62.079,A 180.000,B 0.000,C 180.000} C_DIS
LIN {X 60.982,Y 113.800,Z 62.077,A 180.000,B 0.000,C 180.000} C_DIS
LIN {X 61.059,Y 113.783,Z 62.074,A 180.000,B 0.000,C 180.000} C_DIS
LIN {X 61.213,Y 113.748,Z 62.069,A 180.000,B 0.000,C 180.000} C_DIS
LIN {X 61.366,Y 113.714,Z 62.064,A 180.000,B 0.000,C 180.000} C_DIS
LIN {X 61.520,Y 113.680,Z 62.060,A 180.000,B 0.000,C 180.000} C_DIS
LIN {X 61.673,Y 113.642,Z 62.055,A 180.000,B 0.000,C 180.000} C_DIS
LIN {X 61.824,Y 113.598,Z 62.051,A 180.000,B 0.000,C 180.000} C_DIS
LIN {X 61.976,Y 113.554,Z 62.047,A 180.000,B 0.000,C 180.000} C_DIS
LIN {X 62.127,Y 113.510,Z 62.042,A 180.000,B 0.000,C 180.000} C_DIS
LIN {X 62.278,Y 113.466,Z 62.039,A 180.000,B 0.000,C 180.000} C_DIS
LIN {X 62.428,Y 113.419,Z 62.035,A 180.000,B 0.000,C 180.000} C_DIS
LIN {X 62.576,Y 113.366,Z 62.031,A 180.000,B 0.000,C 180.000} C_DIS
LIN {X 62.725,Y 113.312,Z 62.028,A 180.000,B 0.000,C 180.000} C_DIS
LIN {X 62.873,Y 113.259,Z 62.024,A 180.000,B 0.000,C 180.000} C_DIS
LIN {X 63.021,Y 113.206,Z 62.021,A 180.000,B 0.000,C 180.000} C_DIS
LIN {X 63.168,Y 113.149,Z 62.019,A 180.000,B 0.000,C 180.000} C_DIS
LIN {X 63.313,Y 113.087,Z 62.016,A 180.000,B 0.000,C 180.000} C_DIS
LIN {X 63.602,Y 112.962,Z 62.011,A 180.000,B 0.000,C 180.000} C_DIS
LIN {X 63.889,Y 112.833,Z 62.007,A 180.000,B 0.000,C 180.000} C_DIS
LIN {X 64.170,Y 112.691,Z 62.004,A 180.000,B 0.000,C 180.000} C_DIS
LIN {X 64.451,Y 112.548,Z 62.002,A 180.000,B 0.000,C 180.000} C_DIS
LIN {X 64.725,Y 112.393,Z 62.000,A 180.000,B 0.000,C 180.000} C_DIS
LIN {X 64.959,Y 112.255,Z 62.000,A 180.000,B 0.000,C 180.000} C_DIS
; Cutting Move Starts
LIN {X 65.075,Y 112.186,Z 62.000,A 180.000,B 0.000,C 180.000} C_DIS
LIN {X 65.231,Y 112.092,Z 62.000,A 180.000,B 0.000,C 180.000} C_DIS
LIN {X 65.254,Y 112.077,Z 62.000,A 180.000,B 0.000,C 180.000} C_DIS
LIN {X 65.433,Y 111.956,Z 62.000,A 180.000,B 0.000,C 180.000} C_DIS
LIN {X 65.791,Y 111.713,Z 62.000,A 180.000,B 0.000,C 180.000} C_DIS
LIN {X 65.969,Y 111.583,Z 62.000,A 180.000,B 0.000,C 180.000} C_DIS
LIN {X 66.327,Y 111.306,Z 62.000,A 180.000,B 0.000,C 180.000} C_DIS
LIN {X 66.465,Y 111.198,Z 62.000,A 180.000,B 0.000,C 180.000} C_DIS
LIN {X 66.506,Y 111.165,Z 62.000,A 180.000,B 0.000,C 180.000} C_DIS
LIN {X 66.672,Y 111.019,Z 62.000,A 180.000,B 0.000,C 180.000} C_DIS
LIN {X 66.875,Y 110.841,Z 62.000,A 180.000,B 0.000,C 180.000} C_DIS
LIN {X 67.042,Y 110.693,Z 62.000,A 180.000,B 0.000,C 180.000} C_DIS
LIN {X 67.077,Y 110.662,Z 62.000,A 180.000,B 0.000,C 180.000} C_DIS
LIN {X 67.221,Y 110.521,Z 62.000,A 180.000,B 0.000,C 180.000} C_DIS
LIN {X 67.578,Y 110.163,Z 62.000,A 180.000,B 0.000,C 180.000} C_DIS
LIN {X 67.616,Y 110.126,Z 62.000,A 180.000,B 0.000,C 180.000} C_DIS
LIN {X 67.757,Y 109.970,Z 62.000,A 180.000,B 0.000,C 180.000} C_DIS
LIN {X 68.115,Y 109.564,Z 62.000,A 180.000,B 0.000,C 180.000} C_DIS
LIN {X 68.241,Y 109.410,Z 62.000,A 180.000,B 0.000,C 180.000} C_DIS
LIN {X 68.518,Y 109.053,Z 62.000,A 180.000,B 0.000,C 180.000} C_DIS
LIN {X 68.651,Y 108.880,Z 62.000,A 180.000,B 0.000,C 180.000} C_DIS
LIN {X 68.655,Y 108.874,Z 62.000,A 180.000,B 0.000,C 180.000} C_DIS
LIN {X 68.778,Y 108.695,Z 62.000,A 180.000,B 0.000,C 180.000} C_DIS
LIN {X 69.021,Y 108.338,Z 62.000,A 180.000,B 0.000,C 180.000} C_DIS
LIN {X 69.137,Y 108.159,Z 62.000,A 180.000,B 0.000,C 180.000} C_DIS
LIN {X 69.454,Y 107.623,Z 62.000,A 180.000,B 0.000,C 180.000} C_DIS
LIN {X 69.545,Y 107.456,Z 62.000,A 180.000,B 0.000,C 180.000} C_DIS
LIN {X 69.733,Y 107.086,Z 62.000,A 180.000,B 0.000,C 180.000} C_DIS
LIN {X 69.824,Y 106.908,Z 62.000,A 180.000,B 0.000,C 180.000} C_DIS
LIN {X 69.902,Y 106.739,Z 62.000,A 180.000,B 0.000,C 180.000} C_DIS
LIN {X 70.139,Y 106.193,Z 62.000,A 180.000,B 0.000,C 180.000} C_DIS
LIN {X 70.208,Y 106.014,Z 62.000,A 180.000,B 0.000,C 180.000} C_DIS
LIN {X 70.401,Y 105.477,Z 62.000,A 180.000,B 0.000,C 180.000} C_DIS
LIN {X 70.439,Y 105.369,Z 62.000,A 180.000,B 0.000,C 180.000} C_DIS
LIN {X 70.460,Y 105.299,Z 62.000,A 180.000,B 0.000,C 180.000} C_DIS
LIN {X 70.617,Y 104.758,Z 62.000,A 180.000,B 0.000,C 180.000} C_DIS
LIN {X 70.665,Y 104.584,Z 62.000,A 180.000,B 0.000,C 180.000} C_DIS
LIN {X 70.705,Y 104.405,Z 62.000,A 180.000,B 0.000,C 180.000} C_DIS
LIN {X 70.796,Y 103.999,Z 62.000,A 180.000,B 0.000,C 180.000} C_DIS
LIN {X 70.824,Y 103.869,Z 62.000,A 180.000,B 0.000,C 180.000} C_DIS
LIN {X 70.855,Y 103.690,Z 62.000,A 180.000,B 0.000,C 180.000} C_DIS
LIN {X 70.940,Y 103.153,Z 62.000,A 180.000,B 0.000,C 180.000} C_DIS
LIN {X 70.962,Y 102.975,Z 62.000,A 180.000,B 0.000,C 180.000} C_DIS
LIN {X 71.012,Y 102.438,Z 62.000,A 180.000,B 0.000,C 180.000} C_DIS
LIN {X 71.027,Y 102.260,Z 62.000,A 180.000,B 0.000,C 180.000} C_DIS
LIN {X 71.033,Y 102.081,Z 62.000,A 180.000,B 0.000,C 180.000} C_DIS
LIN {X 71.044,Y 101.723,Z 62.000,A 180.000,B 0.000,C 180.000} C_DIS
LIN {X 71.050,Y 101.545,Z 62.000,A 180.000,B 0.000,C 180.000} C_DIS
LIN {X 71.047,Y 101.366,Z 62.000,A 180.000,B 0.000,C 180.000} C_DIS
LIN {X 71.030,Y 100.829,Z 62.000,A 180.000,B 0.000,C 180.000} C_DIS
LIN {X 71.021,Y 100.651,Z 62.000,A 180.000,B 0.000,C 180.000} C_DIS
LIN {X 71.004,Y 100.472,Z 62.000,A 180.000,B 0.000,C 180.000} C_DIS
LIN {X 70.970,Y 100.114,Z 62.000,A 180.000,B 0.000,C 180.000} C_DIS
LIN {X 70.952,Y 99.936,Z 62.000,A 180.000,B 0.000,C 180.000} C_DIS
LIN {X 70.925,Y 99.757,Z 62.000,A 180.000,B 0.000,C 180.000} C_DIS
LIN {X 70.840,Y 99.221,Z 62.000,A 180.000,B 0.000,C 180.000} C_DIS
LIN {X 70.805,Y 99.042,Z 62.000,A 180.000,B 0.000,C 180.000} C_DIS
LIN {X 70.718,Y 98.654,Z 62.000,A 180.000,B 0.000,C 180.000} C_DIS
LIN {X 70.685,Y 98.505,Z 62.000,A 180.000,B 0.000,C 180.000} C_DIS
LIN {X 70.642,Y 98.327,Z 62.000,A 180.000,B 0.000,C 180.000} C_DIS
LIN {X 70.617,Y 98.242,Z 62.000,A 180.000,B 0.000,C 180.000} C_DIS
LIN {X 70.486,Y 97.790,Z 62.000,A 180.000,B 0.000,C 180.000} C_DIS
LIN {X 70.439,Y 97.631,Z 62.000,A 180.000,B 0.000,C 180.000} C_DIS
LIN {X 70.432,Y 97.612,Z 62.000,A 180.000,B 0.000,C 180.000} C_DIS
LIN {X 70.369,Y 97.433,Z 62.000,A 180.000,B 0.000,C 180.000} C_DIS
LIN {X 70.240,Y 97.075,Z 62.000,A 180.000,B 0.000,C 180.000} C_DIS
LIN {X 70.175,Y 96.897,Z 62.000,A 180.000,B 0.000,C 180.000} C_DIS
LIN {X 70.100,Y 96.718,Z 62.000,A 180.000,B 0.000,C 180.000} C_DIS
LIN {X 69.902,Y 96.261,Z 62.000,A 180.000,B 0.000,C 180.000} C_DIS
LIN {X 69.867,Y 96.181,Z 62.000,A 180.000,B 0.000,C 180.000} C_DIS
LIN {X 69.779,Y 96.003,Z 62.000,A 180.000,B 0.000,C 180.000} C_DIS
LIN {X 69.545,Y 95.544,Z 62.000,A 180.000,B 0.000,C 180.000} C_DIS
LIN {X 69.504,Y 95.466,Z 62.000,A 180.000,B 0.000,C 180.000} C_DIS
LIN {X 69.401,Y 95.288,Z 62.000,A 180.000,B 0.000,C 180.000} C_DIS
LIN {X 69.187,Y 94.927,Z 62.000,A 180.000,B 0.000,C 180.000} C_DIS
LIN {X 69.081,Y 94.751,Z 62.000,A 180.000,B 0.000,C 180.000} C_DIS
LIN {X 69.008,Y 94.644,Z 62.000,A 180.000,B 0.000,C 180.000} C_DIS
LIN {X 68.717,Y 94.215,Z 62.000,A 180.000,B 0.000,C 180.000} C_DIS
LIN {X 68.651,Y 94.120,Z 62.000,A 180.000,B 0.000,C 180.000} C_DIS
LIN {X 68.587,Y 94.036,Z 62.000,A 180.000,B 0.000,C 180.000} C_DIS
LIN {X 68.293,Y 93.657,Z 62.000,A 180.000,B 0.000,C 180.000} C_DIS
LIN {X 68.170,Y 93.500,Z 62.000,A 180.000,B 0.000,C 180.000} C_DIS
LIN {X 68.115,Y 93.436,Z 62.000,A 180.000,B 0.000,C 180.000} C_DIS
LIN {X 67.698,Y 92.964,Z 62.000,A 180.000,B 0.000,C 180.000} C_DIS
LIN {X 67.578,Y 92.837,Z 62.000,A 180.000,B 0.000,C 180.000} C_DIS
LIN {X 67.169,Y 92.427,Z 62.000,A 180.000,B 0.000,C 180.000} C_DIS
LIN {X 67.042,Y 92.307,Z 62.000,A 180.000,B 0.000,C 180.000} C_DIS
LIN {X 66.976,Y 92.249,Z 62.000,A 180.000,B 0.000,C 180.000} C_DIS
LIN {X 66.571,Y 91.891,Z 62.000,A 180.000,B 0.000,C 180.000} C_DIS
LIN {X 66.506,Y 91.835,Z 62.000,A 180.000,B 0.000,C 180.000} C_DIS
LIN {X 66.350,Y 91.712,Z 62.000,A 180.000,B 0.000,C 180.000} C_DIS
LIN {X 65.969,Y 91.417,Z 62.000,A 180.000,B 0.000,C 180.000} C_DIS
LIN {X 65.887,Y 91.355,Z 62.000,A 180.000,B 0.000,C 180.000} C_DIS
LIN {X 65.791,Y 91.287,Z 62.000,A 180.000,B 0.000,C 180.000} C_DIS
LIN {X 65.364,Y 90.997,Z 62.000,A 180.000,B 0.000,C 180.000} C_DIS
LIN {X 65.254,Y 90.923,Z 62.000,A 180.000,B 0.000,C 180.000} C_DIS
LIN {X 65.083,Y 90.818,Z 62.000,A 180.000,B 0.000,C 180.000} C_DIS
LIN {X 64.718,Y 90.603,Z 62.000,A 180.000,B 0.000,C 180.000} C_DIS
LIN {X 64.539,Y 90.499,Z 62.000,A 180.000,B 0.000,C 180.000} C_DIS
LIN {X 64.467,Y 90.461,Z 62.000,A 180.000,B 0.000,C 180.000} C_DIS
LIN {X 64.003,Y 90.224,Z 62.000,A 180.000,B 0.000,C 180.000} C_DIS
LIN {X 63.824,Y 90.135,Z 62.000,A 180.000,B 0.000,C 180.000} C_DIS
LIN {X 63.752,Y 90.103,Z 62.000,A 180.000,B 0.000,C 180.000} C_DIS
LIN {X 63.288,Y 89.903,Z 62.000,A 180.000,B 0.000,C 180.000} C_DIS
LIN {X 63.109,Y 89.827,Z 62.000,A 180.000,B 0.000,C 180.000} C_DIS
LIN {X 62.930,Y 89.762,Z 62.000,A 180.000,B 0.000,C 180.000} C_DIS
LIN {X 62.573,Y 89.633,Z 62.000,A 180.000,B 0.000,C 180.000} C_DIS
LIN {X 62.394,Y 89.569,Z 62.000,A 180.000,B 0.000,C 180.000} C_DIS
LIN {X 62.387,Y 89.567,Z 62.000,A 180.000,B 0.000,C 180.000} C_DIS
LIN {X 62.215,Y 89.516,Z 62.000,A 180.000,B 0.000,C 180.000} C_DIS
LIN {X 61.777,Y 89.388,Z 62.000,A 180.000,B 0.000,C 180.000} C_DIS
LIN {X 61.679,Y 89.360,Z 62.000,A 180.000,B 0.000,C 180.000} C_DIS
LIN {X 61.500,Y 89.316,Z 62.000,A 180.000,B 0.000,C 180.000} C_DIS
LIN {X 60.964,Y 89.196,Z 62.000,A 180.000,B 0.000,C 180.000} C_DIS
LIN {X 60.785,Y 89.161,Z 62.000,A 180.000,B 0.000,C 180.000} C_DIS
LIN {X 60.606,Y 89.132,Z 62.000,A 180.000,B 0.000,C 180.000} C_DIS
LIN {X 60.249,Y 89.076,Z 62.000,A 180.000,B 0.000,C 180.000} C_DIS
LIN {X 60.070,Y 89.049,Z 62.000,A 180.000,B 0.000,C 180.000} C_DIS
LIN {X 59.892,Y 89.031,Z 62.000,A 180.000,B 0.000,C 180.000} C_DIS
LIN {X 59.534,Y 88.997,Z 62.000,A 180.000,B 0.000,C 180.000} C_DIS
LIN {X 59.355,Y 88.980,Z 62.000,A 180.000,B 0.000,C 180.000} C_DIS
LIN {X 59.176,Y 88.970,Z 62.000,A 180.000,B 0.000,C 180.000} C_DIS
LIN {X 58.640,Y 88.953,Z 62.000,A 180.000,B 0.000,C 180.000} C_DIS
LIN {X 58.461,Y 88.950,Z 62.000,A 180.000,B 0.000,C 180.000} C_DIS
LIN {X 58.282,Y 88.956,Z 62.000,A 180.000,B 0.000,C 180.000} C_DIS
LIN {X 57.925,Y 88.967,Z 62.000,A 180.000,B 0.000,C 180.000} C_DIS
LIN {X 57.746,Y 88.973,Z 62.000,A 180.000,B 0.000,C 180.000} C_DIS
LIN {X 57.567,Y 88.987,Z 62.000,A 180.000,B 0.000,C 180.000} C_DIS
LIN {X 57.031,Y 89.038,Z 62.000,A 180.000,B 0.000,C 180.000} C_DIS
LIN {X 56.852,Y 89.060,Z 62.000,A 180.000,B 0.000,C 180.000} C_DIS
LIN {X 56.316,Y 89.145,Z 62.000,A 180.000,B 0.000,C 180.000} C_DIS
LIN {X 56.137,Y 89.174,Z 62.000,A 180.000,B 0.000,C 180.000} C_DIS
LIN {X 55.977,Y 89.209,Z 62.000,A 180.000,B 0.000,C 180.000} C_DIS
LIN {X 55.601,Y 89.293,Z 62.000,A 180.000,B 0.000,C 180.000} C_DIS
LIN {X 55.422,Y 89.334,Z 62.000,A 180.000,B 0.000,C 180.000} C_DIS
LIN {X 55.243,Y 89.382,Z 62.000,A 180.000,B 0.000,C 180.000} C_DIS
LIN {X 54.707,Y 89.538,Z 62.000,A 180.000,B 0.000,C 180.000} C_DIS
LIN {X 54.613,Y 89.567,Z 62.000,A 180.000,B 0.000,C 180.000} C_DIS
LIN {X 54.528,Y 89.597,Z 62.000,A 180.000,B 0.000,C 180.000} C_DIS
LIN {X 53.992,Y 89.790,Z 62.000,A 180.000,B 0.000,C 180.000} C_DIS
LIN {X 53.813,Y 89.859,Z 62.000,A 180.000,B 0.000,C 180.000} C_DIS
LIN {X 53.455,Y 90.014,Z 62.000,A 180.000,B 0.000,C 180.000} C_DIS
LIN {X 53.248,Y 90.103,Z 62.000,A 180.000,B 0.000,C 180.000} C_DIS
LIN {X 53.098,Y 90.173,Z 62.000,A 180.000,B 0.000,C 180.000} C_DIS
LIN {X 52.919,Y 90.264,Z 62.000,A 180.000,B 0.000,C 180.000} C_DIS
LIN {X 52.533,Y 90.461,Z 62.000,A 180.000,B 0.000,C 180.000} C_DIS
LIN {X 52.383,Y 90.543,Z 62.000,A 180.000,B 0.000,C 180.000} C_DIS
LIN {X 51.847,Y 90.860,Z 62.000,A 180.000,B 0.000,C 180.000} C_DIS
LIN {X 51.668,Y 90.975,Z 62.000,A 180.000,B 0.000,C 180.000} C_DIS
LIN {X 51.310,Y 91.218,Z 62.000,A 180.000,B 0.000,C 180.000} C_DIS
LIN {X 51.131,Y 91.341,Z 62.000,A 180.000,B 0.000,C 180.000} C_DIS
LIN {X 51.113,Y 91.355,Z 62.000,A 180.000,B 0.000,C 180.000} C_DIS
LIN {X 50.953,Y 91.478,Z 62.000,A 180.000,B 0.000,C 180.000} C_DIS
LIN {X 50.595,Y 91.755,Z 62.000,A 180.000,B 0.000,C 180.000} C_DIS
LIN {X 50.429,Y 91.891,Z 62.000,A 180.000,B 0.000,C 180.000} C_DIS
LIN {X 50.024,Y 92.249,Z 62.000,A 180.000,B 0.000,C 180.000} C_DIS
LIN {X 49.880,Y 92.379,Z 62.000,A 180.000,B 0.000,C 180.000} C_DIS
LIN {X 49.831,Y 92.427,Z 62.000,A 180.000,B 0.000,C 180.000} C_DIS
LIN {X 49.474,Y 92.785,Z 62.000,A 180.000,B 0.000,C 180.000} C_DIS
LIN {X 49.344,Y 92.917,Z 62.000,A 180.000,B 0.000,C 180.000} C_DIS
LIN {X 49.302,Y 92.964,Z 62.000,A 180.000,B 0.000,C 180.000} C_DIS
LIN {X 48.986,Y 93.321,Z 62.000,A 180.000,B 0.000,C 180.000} C_DIS
LIN {X 48.830,Y 93.500,Z 62.000,A 180.000,B 0.000,C 180.000} C_DIS
LIN {X 48.807,Y 93.528,Z 62.000,A 180.000,B 0.000,C 180.000} C_DIS
LIN {X 48.690,Y 93.679,Z 62.000,A 180.000,B 0.000,C 180.000} C_DIS
LIN {X 48.413,Y 94.036,Z 62.000,A 180.000,B 0.000,C 180.000} C_DIS
LIN {X 48.283,Y 94.215,Z 62.000,A 180.000,B 0.000,C 180.000} C_DIS
LIN {X 48.040,Y 94.573,Z 62.000,A 180.000,B 0.000,C 180.000} C_DIS
LIN {X 47.919,Y 94.751,Z 62.000,A 180.000,B 0.000,C 180.000} C_DIS
LIN {X 47.914,Y 94.760,Z 62.000,A 180.000,B 0.000,C 180.000} C_DIS
LIN {X 47.811,Y 94.930,Z 62.000,A 180.000,B 0.000,C 180.000} C_DIS
LIN {X 47.556,Y 95.361,Z 62.000,A 180.000,B 0.000,C 180.000} C_DIS
LIN {X 47.496,Y 95.466,Z 62.000,A 180.000,B 0.000,C 180.000} C_DIS
LIN {X 47.404,Y 95.645,Z 62.000,A 180.000,B 0.000,C 180.000} C_DIS
LIN {X 47.198,Y 96.048,Z 62.000,A 180.000,B 0.000,C 180.000} C_DIS
LIN {X 47.133,Y 96.181,Z 62.000,A 180.000,B 0.000,C 180.000} C_DIS
LIN {X 47.055,Y 96.360,Z 62.000,A 180.000,B 0.000,C 180.000} C_DIS
LIN {X 46.900,Y 96.718,Z 62.000,A 180.000,B 0.000,C 180.000} C_DIS
LIN {X 46.841,Y 96.856,Z 62.000,A 180.000,B 0.000,C 180.000} C_DIS
LIN {X 46.825,Y 96.897,Z 62.000,A 180.000,B 0.000,C 180.000} C_DIS
LIN {X 46.760,Y 97.075,Z 62.000,A 180.000,B 0.000,C 180.000} C_DIS
LIN {X 46.631,Y 97.433,Z 62.000,A 180.000,B 0.000,C 180.000} C_DIS
LIN {X 46.568,Y 97.612,Z 62.000,A 180.000,B 0.000,C 180.000} C_DIS
LIN {X 46.514,Y 97.790,Z 62.000,A 180.000,B 0.000,C 180.000} C_DIS
LIN {X 46.410,Y 98.148,Z 62.000,A 180.000,B 0.000,C 180.000} C_DIS
LIN {X 46.358,Y 98.327,Z 62.000,A 180.000,B 0.000,C 180.000} C_DIS
LIN {X 46.315,Y 98.505,Z 62.000,A 180.000,B 0.000,C 180.000} C_DIS
LIN {X 46.195,Y 99.042,Z 62.000,A 180.000,B 0.000,C 180.000} C_DIS
LIN {X 46.160,Y 99.221,Z 62.000,A 180.000,B 0.000,C 180.000} C_DIS
LIN {X 46.126,Y 99.434,Z 62.000,A 180.000,B 0.000,C 180.000} C_DIS
LIN {X 46.075,Y 99.757,Z 62.000,A 180.000,B 0.000,C 180.000} C_DIS
LIN {X 46.048,Y 99.936,Z 62.000,A 180.000,B 0.000,C 180.000} C_DIS
LIN {X 46.030,Y 100.114,Z 62.000,A 180.000,B 0.000,C 180.000} C_DIS
LIN {X 45.996,Y 100.472,Z 62.000,A 180.000,B 0.000,C 180.000} C_DIS
LIN {X 45.979,Y 100.651,Z 62.000,A 180.000,B 0.000,C 180.000} C_DIS
LIN {X 45.970,Y 100.829,Z 62.000,A 180.000,B 0.000,C 180.000} C_DIS
LIN {X 45.953,Y 101.366,Z 62.000,A 180.000,B 0.000,C 180.000} C_DIS
LIN {X 45.950,Y 101.545,Z 62.000,A 180.000,B 0.000,C 180.000} C_DIS
LIN {X 45.956,Y 101.723,Z 62.000,A 180.000,B 0.000,C 180.000} C_DIS
LIN {X 45.967,Y 102.081,Z 62.000,A 180.000,B 0.000,C 180.000} C_DIS
LIN {X 45.973,Y 102.260,Z 62.000,A 180.000,B 0.000,C 180.000} C_DIS
LIN {X 45.988,Y 102.438,Z 62.000,A 180.000,B 0.000,C 180.000} C_DIS
LIN {X 46.038,Y 102.975,Z 62.000,A 180.000,B 0.000,C 180.000} C_DIS
LIN {X 46.060,Y 103.153,Z 62.000,A 180.000,B 0.000,C 180.000} C_DIS
LIN {X 46.145,Y 103.690,Z 62.000,A 180.000,B 0.000,C 180.000} C_DIS
LIN {X 46.176,Y 103.869,Z 62.000,A 180.000,B 0.000,C 180.000} C_DIS
LIN {X 46.215,Y 104.047,Z 62.000,A 180.000,B 0.000,C 180.000} C_DIS
LIN {X 46.305,Y 104.449,Z 62.000,A 180.000,B 0.000,C 180.000} C_DIS
LIN {X 46.335,Y 104.584,Z 62.000,A 180.000,B 0.000,C 180.000} C_DIS
LIN {X 46.384,Y 104.762,Z 62.000,A 180.000,B 0.000,C 180.000} C_DIS
LIN {X 46.540,Y 105.299,Z 62.000,A 180.000,B 0.000,C 180.000} C_DIS
LIN {X 46.599,Y 105.477,Z 62.000,A 180.000,B 0.000,C 180.000} C_DIS
LIN {X 46.792,Y 106.014,Z 62.000,A 180.000,B 0.000,C 180.000} C_DIS
LIN {X 46.841,Y 106.144,Z 62.000,A 180.000,B 0.000,C 180.000} C_DIS
LIN {X 46.861,Y 106.193,Z 62.000,A 180.000,B 0.000,C 180.000} C_DIS
LIN {X 47.093,Y 106.729,Z 62.000,A 180.000,B 0.000,C 180.000} C_DIS
LIN {X 47.176,Y 106.908,Z 62.000,A 180.000,B 0.000,C 180.000} C_DIS
LIN {X 47.198,Y 106.952,Z 62.000,A 180.000,B 0.000,C 180.000} C_DIS
LIN {X 47.449,Y 107.444,Z 62.000,A 180.000,B 0.000,C 180.000} C_DIS
LIN {X 47.546,Y 107.623,Z 62.000,A 180.000,B 0.000,C 180.000} C_DIS
LIN {X 47.863,Y 108.159,Z 62.000,A 180.000,B 0.000,C 180.000} C_DIS
LIN {X 47.914,Y 108.240,Z 62.000,A 180.000,B 0.000,C 180.000} C_DIS
LIN {X 47.979,Y 108.338,Z 62.000,A 180.000,B 0.000,C 180.000} C_DIS
LIN {X 48.271,Y 108.767,Z 62.000,A 180.000,B 0.000,C 180.000} C_DIS
LIN {X 48.345,Y 108.874,Z 62.000,A 180.000,B 0.000,C 180.000} C_DIS
LIN {X 48.450,Y 109.012,Z 62.000,A 180.000,B 0.000,C 180.000} C_DIS
LIN {X 48.759,Y 109.410,Z 62.000,A 180.000,B 0.000,C 180.000} C_DIS
LIN {X 48.807,Y 109.472,Z 62.000,A 180.000,B 0.000,C 180.000} C_DIS
LIN {X 48.907,Y 109.589,Z 62.000,A 180.000,B 0.000,C 180.000} C_DIS
LIN {X 49.223,Y 109.947,Z 62.000,A 180.000,B 0.000,C 180.000} C_DIS
LIN {X 49.344,Y 110.083,Z 62.000,A 180.000,B 0.000,C 180.000} C_DIS
LIN {X 49.384,Y 110.126,Z 62.000,A 180.000,B 0.000,C 180.000} C_DIS
LIN {X 49.523,Y 110.264,Z 62.000,A 180.000,B 0.000,C 180.000} C_DIS
LIN {X 49.742,Y 110.483,Z 62.000,A 180.000,B 0.000,C 180.000} C_DIS
LIN {X 49.880,Y 110.621,Z 62.000,A 180.000,B 0.000,C 180.000} C_DIS
LIN {X 49.923,Y 110.662,Z 62.000,A 180.000,B 0.000,C 180.000} C_DIS
LIN {X 50.059,Y 110.782,Z 62.000,A 180.000,B 0.000,C 180.000} C_DIS
LIN {X 50.416,Y 111.098,Z 62.000,A 180.000,B 0.000,C 180.000} C_DIS
LIN {X 50.535,Y 111.198,Z 62.000,A 180.000,B 0.000,C 180.000} C_DIS
LIN {X 50.595,Y 111.245,Z 62.000,A 180.000,B 0.000,C 180.000} C_DIS
LIN {X 50.996,Y 111.556,Z 62.000,A 180.000,B 0.000,C 180.000} C_DIS
LIN {X 51.131,Y 111.659,Z 62.000,A 180.000,B 0.000,C 180.000} C_DIS
LIN {X 51.241,Y 111.734,Z 62.000,A 180.000,B 0.000,C 180.000} C_DIS
LIN {X 51.668,Y 112.025,Z 62.000,A 180.000,B 0.000,C 180.000} C_DIS
LIN {X 51.769,Y 112.092,Z 62.000,A 180.000,B 0.000,C 180.000} C_DIS
LIN {X 51.847,Y 112.140,Z 62.000,A 180.000,B 0.000,C 180.000} C_DIS
LIN {X 52.383,Y 112.457,Z 62.000,A 180.000,B 0.000,C 180.000} C_DIS
LIN {X 52.562,Y 112.554,Z 62.000,A 180.000,B 0.000,C 180.000} C_DIS
LIN {X 53.059,Y 112.807,Z 62.000,A 180.000,B 0.000,C 180.000} C_DIS
LIN {X 53.098,Y 112.827,Z 62.000,A 180.000,B 0.000,C 180.000} C_DIS
LIN {X 53.277,Y 112.909,Z 62.000,A 180.000,B 0.000,C 180.000} C_DIS
LIN {X 53.813,Y 113.141,Z 62.000,A 180.000,B 0.000,C 180.000} C_DIS
LIN {X 53.870,Y 113.165,Z 62.000,A 180.000,B 0.000,C 180.000} C_DIS
LIN {X 53.992,Y 113.210,Z 62.000,A 180.000,B 0.000,C 180.000} C_DIS
LIN {X 54.528,Y 113.403,Z 62.000,A 180.000,B 0.000,C 180.000} C_DIS
LIN {X 54.707,Y 113.462,Z 62.000,A 180.000,B 0.000,C 180.000} C_DIS
LIN {X 55.243,Y 113.618,Z 62.000,A 180.000,B 0.000,C 180.000} C_DIS
LIN {X 55.422,Y 113.666,Z 62.000,A 180.000,B 0.000,C 180.000} C_DIS
LIN {X 55.575,Y 113.701,Z 62.000,A 180.000,B 0.000,C 180.000} C_DIS
LIN {X 55.958,Y 113.786,Z 62.000,A 180.000,B 0.000,C 180.000} C_DIS
LIN {X 56.137,Y 113.826,Z 62.000,A 180.000,B 0.000,C 180.000} C_DIS
LIN {X 56.316,Y 113.855,Z 62.000,A 180.000,B 0.000,C 180.000} C_DIS
LIN {X 56.852,Y 113.940,Z 62.000,A 180.000,B 0.000,C 180.000} C_DIS
LIN {X 57.031,Y 113.962,Z 62.000,A 180.000,B 0.000,C 180.000} C_DIS
LIN {X 57.567,Y 114.013,Z 62.000,A 180.000,B 0.000,C 180.000} C_DIS
LIN {X 57.746,Y 114.027,Z 62.000,A 180.000,B 0.000,C 180.000} C_DIS
LIN {X 57.925,Y 114.033,Z 62.000,A 180.000,B 0.000,C 180.000} C_DIS
LIN {X 58.282,Y 114.044,Z 62.000,A 180.000,B 0.000,C 180.000} C_DIS
LIN {X 58.461,Y 114.050,Z 62.000,A 180.000,B 0.000,C 180.000} C_DIS
LIN {X 58.640,Y 114.047,Z 62.000,A 180.000,B 0.000,C 180.000} C_DIS
LIN {X 59.176,Y 114.030,Z 62.000,A 180.000,B 0.000,C 180.000} C_DIS
LIN {X 59.355,Y 114.020,Z 62.000,A 180.000,B 0.000,C 180.000} C_DIS
LIN {X 59.534,Y 114.003,Z 62.000,A 180.000,B 0.000,C 180.000} C_DIS
LIN {X 59.891,Y 113.969,Z 62.000,A 180.000,B 0.000,C 180.000} C_DIS
LIN {X 60.070,Y 113.951,Z 62.000,A 180.000,B 0.000,C 180.000} C_DIS
LIN {X 60.249,Y 113.924,Z 62.000,A 180.000,B 0.000,C 180.000} C_DIS
LIN {X 60.606,Y 113.868,Z 62.000,A 180.000,B 0.000,C 180.000} C_DIS
LIN {X 60.785,Y 113.839,Z 62.000,A 180.000,B 0.000,C 180.000} C_DIS
LIN {X 60.964,Y 113.804,Z 62.000,A 180.000,B 0.000,C 180.000} C_DIS
LIN {X 61.500,Y 113.684,Z 62.000,A 180.000,B 0.000,C 180.000} C_DIS
LIN {X 61.679,Y 113.640,Z 62.000,A 180.000,B 0.000,C 180.000} C_DIS
LIN {X 61.858,Y 113.588,Z 62.000,A 180.000,B 0.000,C 180.000} C_DIS
LIN {X 62.215,Y 113.484,Z 62.000,A 180.000,B 0.000,C 180.000} C_DIS
LIN {X 62.394,Y 113.431,Z 62.000,A 180.000,B 0.000,C 180.000} C_DIS
LIN {X 62.573,Y 113.367,Z 62.000,A 180.000,B 0.000,C 180.000} C_DIS
LIN {X 62.930,Y 113.238,Z 62.000,A 180.000,B 0.000,C 180.000} C_DIS
LIN {X 63.109,Y 113.173,Z 62.000,A 180.000,B 0.000,C 180.000} C_DIS
LIN {X 63.130,Y 113.165,Z 62.000,A 180.000,B 0.000,C 180.000} C_DIS
LIN {X 63.288,Y 113.097,Z 62.000,A 180.000,B 0.000,C 180.000} C_DIS
LIN {X 63.645,Y 112.943,Z 62.000,A 180.000,B 0.000,C 180.000} C_DIS
LIN {X 63.824,Y 112.865,Z 62.000,A 180.000,B 0.000,C 180.000} C_DIS
LIN {X 63.941,Y 112.807,Z 62.000,A 180.000,B 0.000,C 180.000} C_DIS
LIN {X 64.360,Y 112.594,Z 62.000,A 180.000,B 0.000,C 180.000} C_DIS
LIN {X 64.539,Y 112.501,Z 62.000,A 180.000,B 0.000,C 180.000} C_DIS
LIN {X 64.630,Y 112.450,Z 62.000,A 180.000,B 0.000,C 180.000} C_DIS
LIN {X 64.959,Y 112.255,Z 62.000,A 180.000,B 0.000,C 180.000} C_DIS
; Lead Out Move Starts
LIN {X 65.545,Y 112.312,Z 62.000,A 180.000,B 0.000,C 180.000} C_DIS
LIN {X 65.671,Y 112.888,Z 62.000,A 180.000,B 0.000,C 180.000} C_DIS
; Link Move Starts
LIN {X 49.015,Y 150.527,Z 62.000,A 180.000,B 0.000,C 180.000} C_DIS
LIN {X 49.015,Y 150.527,Z 57.550,A 180.000,B 0.000,C 180.000} C_DIS
$VEL.CP=0.01
LIN {X 49.016,Y 150.525,Z 57.507,A 180.000,B 0.000,C 180.000} C_DIS
LIN {X 49.016,Y 150.519,Z 57.465,A 180.000,B 0.000,C 180.000} C_DIS
LIN {X 49.016,Y 150.510,Z 57.423,A 180.000,B 0.000,C 180.000} C_DIS
LIN {X 49.017,Y 150.498,Z 57.382,A 180.000,B 0.000,C 180.000} C_DIS
LIN {X 49.017,Y 150.482,Z 57.343,A 180.000,B 0.000,C 180.000} C_DIS
LIN {X 49.019,Y 150.463,Z 57.305,A 180.000,B 0.000,C 180.000} C_DIS
LIN {X 49.020,Y 150.440,Z 57.268,A 180.000,B 0.000,C 180.000} C_DIS
LIN {X 49.022,Y 150.415,Z 57.234,A 180.000,B 0.000,C 180.000} C_DIS
LIN {X 49.024,Y 150.387,Z 57.202,A 180.000,B 0.000,C 180.000} C_DIS
LIN {X 49.027,Y 150.356,Z 57.173,A 180.000,B 0.000,C 180.000} C_DIS
LIN {X 49.031,Y 150.323,Z 57.146,A 180.000,B 0.000,C 180.000} C_DIS
LIN {X 49.036,Y 150.288,Z 57.123,A 180.000,B 0.000,C 180.000} C_DIS
LIN {X 49.041,Y 150.251,Z 57.102,A 180.000,B 0.000,C 180.000} C_DIS
LIN {X 49.047,Y 150.212,Z 57.085,A 180.000,B 0.000,C 180.000} C_DIS
LIN {X 49.054,Y 150.172,Z 57.071,A 180.000,B 0.000,C 180.000} C_DIS
LIN {X 49.062,Y 150.132,Z 57.060,A 180.000,B 0.000,C 180.000} C_DIS
LIN {X 49.071,Y 150.091,Z 57.053,A 180.000,B 0.000,C 180.000} C_DIS
LIN {X 49.081,Y 150.049,Z 57.050,A 180.000,B 0.000,C 180.000} C_DIS
LIN {X 49.756,Y 148.883,Z 57.002,A 180.000,B 0.000,C 180.000} C_DIS
LIN {X 50.958,Y 148.272,Z 56.955,A 180.000,B 0.000,C 180.000} C_DIS
LIN {X 52.299,Y 148.414,Z 56.907,A 180.000,B 0.000,C 180.000} C_DIS
LIN {X 53.346,Y 149.262,Z 56.859,A 180.000,B 0.000,C 180.000} C_DIS
LIN {X 53.763,Y 150.544,Z 56.811,A 180.000,B 0.000,C 180.000} C_DIS
LIN {X 53.415,Y 151.847,Z 56.764,A 180.000,B 0.000,C 180.000} C_DIS
LIN {X 52.414,Y 152.750,Z 56.716,A 180.000,B 0.000,C 180.000} C_DIS
LIN {X 51.083,Y 152.963,Z 56.668,A 180.000,B 0.000,C 180.000} C_DIS
LIN {X 49.851,Y 152.417,Z 56.621,A 180.000,B 0.000,C 180.000} C_DIS
LIN {X 49.114,Y 151.288,Z 56.573,A 180.000,B 0.000,C 180.000} C_DIS
LIN {X 49.110,Y 149.940,Z 56.525,A 180.000,B 0.000,C 180.000} C_DIS
LIN {X 49.840,Y 148.807,Z 56.477,A 180.000,B 0.000,C 180.000} C_DIS
LIN {X 51.070,Y 148.254,Z 56.430,A 180.000,B 0.000,C 180.000} C_DIS
LIN {X 52.402,Y 148.459,Z 56.382,A 180.000,B 0.000,C 180.000} C_DIS
LIN {X 53.408,Y 149.357,Z 56.334,A 180.000,B 0.000,C 180.000} C_DIS
LIN {X 53.764,Y 150.657,Z 56.287,A 180.000,B 0.000,C 180.000} C_DIS
LIN {X 53.354,Y 151.942,Z 56.239,A 180.000,B 0.000,C 180.000} C_DIS
LIN {X 52.311,Y 152.796,Z 56.191,A 180.000,B 0.000,C 180.000} C_DIS
LIN {X 50.971,Y 152.945,Z 56.143,A 180.000,B 0.000,C 180.000} C_DIS
LIN {X 49.766,Y 152.341,Z 56.096,A 180.000,B 0.000,C 180.000} C_DIS
LIN {X 49.084,Y 151.179,Z 56.048,A 180.000,B 0.000,C 180.000} C_DIS
LIN {X 49.144,Y 149.832,Z 56.000,A 180.000,B 0.000,C 180.000} C_DIS
LIN {X 49.150,Y 149.816,Z 56.000,A 180.000,B 0.000,C 180.000} C_DIS
; Lead In Move Starts
LIN {X 49.235,Y 149.575,Z 56.000,A 180.000,B 0.000,C 180.000} C_DIS
LIN {X 49.932,Y 148.560,Z 56.000,A 180.000,B 0.000,C 180.000} C_DIS
LIN {X 51.044,Y 148.029,Z 56.000,A 180.000,B 0.000,C 180.000} C_DIS
LIN {X 52.272,Y 148.125,Z 56.000,A 180.000,B 0.000,C 180.000} C_DIS
; Cutting Move Starts
$VEL.CP=0.02
LIN {X 53.277,Y 148.480,Z 56.000,A 180.000,B 0.000,C 180.000} C_DIS
LIN {X 53.455,Y 148.540,Z 56.000,A 180.000,B 0.000,C 180.000} C_DIS
LIN {X 54.290,Y 148.813,Z 56.000,A 180.000,B 0.000,C 180.000} C_DIS
LIN {X 54.886,Y 149.008,Z 56.000,A 180.000,B 0.000,C 180.000} C_DIS
LIN {X 55.064,Y 149.065,Z 56.000,A 180.000,B 0.000,C 180.000} C_DIS
LIN {X 56.495,Y 149.497,Z 56.000,A 180.000,B 0.000,C 180.000} C_DIS
LIN {X 56.673,Y 149.550,Z 56.000,A 180.000,B 0.000,C 180.000} C_DIS
LIN {X 56.852,Y 149.600,Z 56.000,A 180.000,B 0.000,C 180.000} C_DIS
LIN {X 58.282,Y 149.995,Z 56.000,A 180.000,B 0.000,C 180.000} C_DIS
LIN {X 58.461,Y 150.042,Z 56.000,A 180.000,B 0.000,C 180.000} C_DIS
LIN {X 59.891,Y 150.402,Z 56.000,A 180.000,B 0.000,C 180.000} C_DIS
LIN {X 60.070,Y 150.447,Z 56.000,A 180.000,B 0.000,C 180.000} C_DIS
LIN {X 60.249,Y 150.487,Z 56.000,A 180.000,B 0.000,C 180.000} C_DIS
LIN {X 61.679,Y 150.811,Z 56.000,A 180.000,B 0.000,C 180.000} C_DIS
LIN {X 61.858,Y 150.850,Z 56.000,A 180.000,B 0.000,C 180.000} C_DIS
LIN {X 63.467,Y 151.175,Z 56.000,A 180.000,B 0.000,C 180.000} C_DIS
LIN {X 63.645,Y 151.208,Z 56.000,A 180.000,B 0.000,C 180.000} C_DIS
LIN {X 65.075,Y 151.462,Z 56.000,A 180.000,B 0.000,C 180.000} C_DIS
LIN {X 65.254,Y 151.494,Z 56.000,A 180.000,B 0.000,C 180.000} C_DIS
LIN {X 65.433,Y 151.521,Z 56.000,A 180.000,B 0.000,C 180.000} C_DIS
LIN {X 66.863,Y 151.741,Z 56.000,A 180.000,B 0.000,C 180.000} C_DIS
LIN {X 67.042,Y 151.767,Z 56.000,A 180.000,B 0.000,C 180.000} C_DIS
LIN {X 68.651,Y 151.975,Z 56.000,A 180.000,B 0.000,C 180.000} C_DIS
LIN {X 68.830,Y 151.996,Z 56.000,A 180.000,B 0.000,C 180.000} C_DIS
LIN {X 70.439,Y 152.167,Z 56.000,A 180.000,B 0.000,C 180.000} C_DIS
LIN {X 70.617,Y 152.182,Z 56.000,A 180.000,B 0.000,C 180.000} C_DIS
LIN {X 72.048,Y 152.300,Z 56.000,A 180.000,B 0.000,C 180.000} C_DIS
LIN {X 72.226,Y 152.314,Z 56.000,A 180.000,B 0.000,C 180.000} C_DIS
LIN {X 72.239,Y 152.315,Z 56.000,A 180.000,B 0.000,C 180.000} C_DIS
LIN {X 72.405,Y 152.325,Z 56.000,A 180.000,B 0.000,C 180.000} C_DIS
LIN {X 73.835,Y 152.409,Z 56.000,A 180.000,B 0.000,C 180.000} C_DIS
LIN {X 74.014,Y 152.419,Z 56.000,A 180.000,B 0.000,C 180.000} C_DIS
LIN {X 75.623,Y 152.475,Z 56.000,A 180.000,B 0.000,C 180.000} C_DIS
LIN {X 75.802,Y 152.480,Z 56.000,A 180.000,B 0.000,C 180.000} C_DIS
LIN {X 77.411,Y 152.499,Z 56.000,A 180.000,B 0.000,C 180.000} C_DIS
LIN {X 77.589,Y 152.499,Z 56.000,A 180.000,B 0.000,C 180.000} C_DIS
LIN {X 79.198,Y 152.480,Z 56.000,A 180.000,B 0.000,C 180.000} C_DIS
LIN {X 79.377,Y 152.475,Z 56.000,A 180.000,B 0.000,C 180.000} C_DIS
LIN {X 80.986,Y 152.419,Z 56.000,A 180.000,B 0.000,C 180.000} C_DIS
LIN {X 81.165,Y 152.409,Z 56.000,A 180.000,B 0.000,C 180.000} C_DIS
LIN {X 82.595,Y 152.325,Z 56.000,A 180.000,B 0.000,C 180.000} C_DIS
LIN {X 82.761,Y 152.315,Z 56.000,A 180.000,B 0.000,C 180.000} C_DIS
LIN {X 82.774,Y 152.314,Z 56.000,A 180.000,B 0.000,C 180.000} C_DIS
LIN {X 82.952,Y 152.300,Z 56.000,A 180.000,B 0.000,C 180.000} C_DIS
LIN {X 84.383,Y 152.182,Z 56.000,A 180.000,B 0.000,C 180.000} C_DIS
LIN {X 84.561,Y 152.167,Z 56.000,A 180.000,B 0.000,C 180.000} C_DIS
LIN {X 86.170,Y 151.996,Z 56.000,A 180.000,B 0.000,C 180.000} C_DIS
LIN {X 86.349,Y 151.975,Z 56.000,A 180.000,B 0.000,C 180.000} C_DIS
LIN {X 87.958,Y 151.767,Z 56.000,A 180.000,B 0.000,C 180.000} C_DIS
LIN {X 88.137,Y 151.741,Z 56.000,A 180.000,B 0.000,C 180.000} C_DIS
LIN {X 89.567,Y 151.521,Z 56.000,A 180.000,B 0.000,C 180.000} C_DIS
LIN {X 89.746,Y 151.494,Z 56.000,A 180.000,B 0.000,C 180.000} C_DIS
LIN {X 89.925,Y 151.462,Z 56.000,A 180.000,B 0.000,C 180.000} C_DIS
LIN {X 91.355,Y 151.208,Z 56.000,A 180.000,B 0.000,C 180.000} C_DIS
LIN {X 91.533,Y 151.175,Z 56.000,A 180.000,B 0.000,C 180.000} C_DIS
LIN {X 93.142,Y 150.850,Z 56.000,A 180.000,B 0.000,C 180.000} C_DIS
LIN {X 93.321,Y 150.811,Z 56.000,A 180.000,B 0.000,C 180.000} C_DIS
LIN {X 94.751,Y 150.487,Z 56.000,A 180.000,B 0.000,C 180.000} C_DIS
LIN {X 94.930,Y 150.447,Z 56.000,A 180.000,B 0.000,C 180.000} C_DIS
LIN {X 95.109,Y 150.402,Z 56.000,A 180.000,B 0.000,C 180.000} C_DIS
LIN {X 96.539,Y 150.042,Z 56.000,A 180.000,B 0.000,C 180.000} C_DIS
LIN {X 96.718,Y 149.995,Z 56.000,A 180.000,B 0.000,C 180.000} C_DIS
LIN {X 98.148,Y 149.600,Z 56.000,A 180.000,B 0.000,C 180.000} C_DIS
LIN {X 98.327,Y 149.550,Z 56.000,A 180.000,B 0.000,C 180.000} C_DIS
LIN {X 98.505,Y 149.497,Z 56.000,A 180.000,B 0.000,C 180.000} C_DIS
LIN {X 99.936,Y 149.065,Z 56.000,A 180.000,B 0.000,C 180.000} C_DIS
LIN {X 100.114,Y 149.008,Z 56.000,A 180.000,B 0.000,C 180.000} C_DIS
LIN {X 101.545,Y 148.540,Z 56.000,A 180.000,B 0.000,C 180.000} C_DIS
LIN {X 101.723,Y 148.480,Z 56.000,A 180.000,B 0.000,C 180.000} C_DIS
LIN {X 103.153,Y 147.974,Z 56.000,A 180.000,B 0.000,C 180.000} C_DIS
LIN {X 103.332,Y 147.911,Z 56.000,A 180.000,B 0.000,C 180.000} C_DIS
LIN {X 103.504,Y 147.846,Z 56.000,A 180.000,B 0.000,C 180.000} C_DIS
LIN {X 104.941,Y 147.299,Z 56.000,A 180.000,B 0.000,C 180.000} C_DIS
LIN {X 105.120,Y 147.227,Z 56.000,A 180.000,B 0.000,C 180.000} C_DIS
LIN {X 106.550,Y 146.645,Z 56.000,A 180.000,B 0.000,C 180.000} C_DIS
LIN {X 106.669,Y 146.595,Z 56.000,A 180.000,B 0.000,C 180.000} C_DIS
LIN {X 108.159,Y 145.947,Z 56.000,A 180.000,B 0.000,C 180.000} C_DIS
LIN {X 108.308,Y 145.880,Z 56.000,A 180.000,B 0.000,C 180.000} C_DIS
LIN {X 109.768,Y 145.203,Z 56.000,A 180.000,B 0.000,C 180.000} C_DIS
LIN {X 109.849,Y 145.164,Z 56.000,A 180.000,B 0.000,C 180.000} C_DIS
LIN {X 111.303,Y 144.449,Z 56.000,A 180.000,B 0.000,C 180.000} C_DIS
LIN {X 111.377,Y 144.413,Z 56.000,A 180.000,B 0.000,C 180.000} C_DIS
LIN {X 111.556,Y 144.320,Z 56.000,A 180.000,B 0.000,C 180.000} C_DIS
LIN {X 112.807,Y 143.668,Z 56.000,A 180.000,B 0.000,C 180.000} C_DIS
LIN {X 112.986,Y 143.574,Z 56.000,A 180.000,B 0.000,C 180.000} C_DIS
LIN {X 114.416,Y 142.785,Z 56.000,A 180.000,B 0.000,C 180.000} C_DIS
LIN {X 114.595,Y 142.683,Z 56.000,A 180.000,B 0.000,C 180.000} C_DIS
LIN {X 115.859,Y 141.947,Z 56.000,A 180.000,B 0.000,C 180.000} C_DIS
LIN {X 116.025,Y 141.849,Z 56.000,A 180.000,B 0.000,C 180.000} C_DIS
LIN {X 116.158,Y 141.768,Z 56.000,A 180.000,B 0.000,C 180.000} C_DIS
LIN {X 117.455,Y 140.971,Z 56.000,A 180.000,B 0.000,C 180.000} C_DIS
LIN {X 117.607,Y 140.874,Z 56.000,A 180.000,B 0.000,C 180.000} C_DIS
LIN {X 118.885,Y 140.047,Z 56.000,A 180.000,B 0.000,C 180.000} C_DIS
LIN {X 118.988,Y 139.980,Z 56.000,A 180.000,B 0.000,C 180.000} C_DIS
LIN {X 119.064,Y 139.928,Z 56.000,A 180.000,B 0.000,C 180.000} C_DIS
LIN {X 120.315,Y 139.076,Z 56.000,A 180.000,B 0.000,C 180.000} C_DIS
LIN {X 120.494,Y 138.953,Z 56.000,A 180.000,B 0.000,C 180.000} C_DIS
LIN {X 121.806,Y 138.014,Z 56.000,A 180.000,B 0.000,C 180.000} C_DIS
LIN {X 121.924,Y 137.927,Z 56.000,A 180.000,B 0.000,C 180.000} C_DIS
LIN {X 123.235,Y 136.941,Z 56.000,A 180.000,B 0.000,C 180.000} C_DIS
LIN {X 123.354,Y 136.848,Z 56.000,A 180.000,B 0.000,C 180.000} C_DIS
LIN {X 124.606,Y 135.861,Z 56.000,A 180.000,B 0.000,C 180.000} C_DIS
LIN {X 124.785,Y 135.714,Z 56.000,A 180.000,B 0.000,C 180.000} C_DIS
LIN {X 125.894,Y 134.796,Z 56.000,A 180.000,B 0.000,C 180.000} C_DIS
LIN {X 126.036,Y 134.677,Z 56.000,A 180.000,B 0.000,C 180.000} C_DIS
LIN {X 127.287,Y 133.590,Z 56.000,A 180.000,B 0.000,C 180.000} C_DIS
LIN {X 127.340,Y 133.544,Z 56.000,A 180.000,B 0.000,C 180.000} C_DIS
LIN {X 127.466,Y 133.430,Z 56.000,A 180.000,B 0.000,C 180.000} C_DIS
LIN {X 128.539,Y 132.453,Z 56.000,A 180.000,B 0.000,C 180.000} C_DIS
LIN {X 128.711,Y 132.293,Z 56.000,A 180.000,B 0.000,C 180.000} C_DIS
LIN {X 129.835,Y 131.220,Z 56.000,A 180.000,B 0.000,C 180.000} C_DIS
LIN {X 129.969,Y 131.090,Z 56.000,A 180.000,B 0.000,C 180.000} C_DIS
LIN {X 131.090,Y 129.969,Z 56.000,A 180.000,B 0.000,C 180.000} C_DIS
LIN {X 131.220,Y 129.835,Z 56.000,A 180.000,B 0.000,C 180.000} C_DIS
LIN {X 132.293,Y 128.711,Z 56.000,A 180.000,B 0.000,C 180.000} C_DIS
LIN {X 132.453,Y 128.539,Z 56.000,A 180.000,B 0.000,C 180.000} C_DIS
LIN {X 133.430,Y 127.466,Z 56.000,A 180.000,B 0.000,C 180.000} C_DIS
LIN {X 133.544,Y 127.340,Z 56.000,A 180.000,B 0.000,C 180.000} C_DIS
LIN {X 133.590,Y 127.287,Z 56.000,A 180.000,B 0.000,C 180.000} C_DIS
LIN {X 134.677,Y 126.036,Z 56.000,A 180.000,B 0.000,C 180.000} C_DIS
LIN {X 134.796,Y 125.894,Z 56.000,A 180.000,B 0.000,C 180.000} C_DIS
LIN {X 135.714,Y 124.785,Z 56.000,A 180.000,B 0.000,C 180.000} C_DIS
LIN {X 135.861,Y 124.606,Z 56.000,A 180.000,B 0.000,C 180.000} C_DIS
LIN {X 136.848,Y 123.354,Z 56.000,A 180.000,B 0.000,C 180.000} C_DIS
LIN {X 136.941,Y 123.235,Z 56.000,A 180.000,B 0.000,C 180.000} C_DIS
LIN {X 137.927,Y 121.924,Z 56.000,A 180.000,B 0.000,C 180.000} C_DIS
LIN {X 138.014,Y 121.806,Z 56.000,A 180.000,B 0.000,C 180.000} C_DIS
LIN {X 138.953,Y 120.494,Z 56.000,A 180.000,B 0.000,C 180.000} C_DIS
LIN {X 139.076,Y 120.315,Z 56.000,A 180.000,B 0.000,C 180.000} C_DIS
LIN {X 139.928,Y 119.064,Z 56.000,A 180.000,B 0.000,C 180.000} C_DIS
LIN {X 139.980,Y 118.988,Z 56.000,A 180.000,B 0.000,C 180.000} C_DIS
LIN {X 140.047,Y 118.885,Z 56.000,A 180.000,B 0.000,C 180.000} C_DIS
LIN {X 140.874,Y 117.607,Z 56.000,A 180.000,B 0.000,C 180.000} C_DIS
LIN {X 140.971,Y 117.455,Z 56.000,A 180.000,B 0.000,C 180.000} C_DIS
LIN {X 141.768,Y 116.158,Z 56.000,A 180.000,B 0.000,C 180.000} C_DIS
LIN {X 141.849,Y 116.025,Z 56.000,A 180.000,B 0.000,C 180.000} C_DIS
LIN {X 141.947,Y 115.859,Z 56.000,A 180.000,B 0.000,C 180.000} C_DIS
LIN {X 142.683,Y 114.595,Z 56.000,A 180.000,B 0.000,C 180.000} C_DIS
LIN {X 142.785,Y 114.416,Z 56.000,A 180.000,B 0.000,C 180.000} C_DIS
LIN {X 143.574,Y 112.986,Z 56.000,A 180.000,B 0.000,C 180.000} C_DIS
LIN {X 143.668,Y 112.807,Z 56.000,A 180.000,B 0.000,C 180.000} C_DIS
LIN {X 144.320,Y 111.556,Z 56.000,A 180.000,B 0.000,C 180.000} C_DIS
LIN {X 144.413,Y 111.377,Z 56.000,A 180.000,B 0.000,C 180.000} C_DIS
LIN {X 144.449,Y 111.303,Z 56.000,A 180.000,B 0.000,C 180.000} C_DIS
LIN {X 145.164,Y 109.849,Z 56.000,A 180.000,B 0.000,C 180.000} C_DIS
LIN {X 145.203,Y 109.768,Z 56.000,A 180.000,B 0.000,C 180.000} C_DIS
LIN {X 145.880,Y 108.308,Z 56.000,A 180.000,B 0.000,C 180.000} C_DIS
LIN {X 145.947,Y 108.159,Z 56.000,A 180.000,B 0.000,C 180.000} C_DIS
LIN {X 146.595,Y 106.669,Z 56.000,A 180.000,B 0.000,C 180.000} C_DIS
LIN {X 146.645,Y 106.550,Z 56.000,A 180.000,B 0.000,C 180.000} C_DIS
LIN {X 147.227,Y 105.120,Z 56.000,A 180.000,B 0.000,C 180.000} C_DIS
LIN {X 147.299,Y 104.941,Z 56.000,A 180.000,B 0.000,C 180.000} C_DIS
LIN {X 147.846,Y 103.504,Z 56.000,A 180.000,B 0.000,C 180.000} C_DIS
LIN {X 147.911,Y 103.332,Z 56.000,A 180.000,B 0.000,C 180.000} C_DIS
LIN {X 147.974,Y 103.153,Z 56.000,A 180.000,B 0.000,C 180.000} C_DIS
LIN {X 148.480,Y 101.723,Z 56.000,A 180.000,B 0.000,C 180.000} C_DIS
LIN {X 148.540,Y 101.545,Z 56.000,A 180.000,B 0.000,C 180.000} C_DIS
LIN {X 149.008,Y 100.114,Z 56.000,A 180.000,B 0.000,C 180.000} C_DIS
LIN {X 149.065,Y 99.936,Z 56.000,A 180.000,B 0.000,C 180.000} C_DIS
LIN {X 149.497,Y 98.505,Z 56.000,A 180.000,B 0.000,C 180.000} C_DIS
LIN {X 149.550,Y 98.327,Z 56.000,A 180.000,B 0.000,C 180.000} C_DIS
LIN {X 149.600,Y 98.148,Z 56.000,A 180.000,B 0.000,C 180.000} C_DIS
LIN {X 149.995,Y 96.718,Z 56.000,A 180.000,B 0.000,C 180.000} C_DIS
LIN {X 150.042,Y 96.539,Z 56.000,A 180.000,B 0.000,C 180.000} C_DIS
LIN {X 150.402,Y 95.109,Z 56.000,A 180.000,B 0.000,C 180.000} C_DIS
LIN {X 150.447,Y 94.930,Z 56.000,A 180.000,B 0.000,C 180.000} C_DIS
LIN {X 150.487,Y 94.751,Z 56.000,A 180.000,B 0.000,C 180.000} C_DIS
LIN {X 150.811,Y 93.321,Z 56.000,A 180.000,B 0.000,C 180.000} C_DIS
LIN {X 150.850,Y 93.142,Z 56.000,A 180.000,B 0.000,C 180.000} C_DIS
LIN {X 151.175,Y 91.533,Z 56.000,A 180.000,B 0.000,C 180.000} C_DIS
LIN {X 151.208,Y 91.355,Z 56.000,A 180.000,B 0.000,C 180.000} C_DIS
LIN {X 151.462,Y 89.925,Z 56.000,A 180.000,B 0.000,C 180.000} C_DIS
LIN {X 151.494,Y 89.746,Z 56.000,A 180.000,B 0.000,C 180.000} C_DIS
LIN {X 151.521,Y 89.567,Z 56.000,A 180.000,B 0.000,C 180.000} C_DIS
LIN {X 151.741,Y 88.137,Z 56.000,A 180.000,B 0.000,C 180.000} C_DIS
LIN {X 151.767,Y 87.958,Z 56.000,A 180.000,B 0.000,C 180.000} C_DIS
LIN {X 151.975,Y 86.349,Z 56.000,A 180.000,B 0.000,C 180.000} C_DIS
LIN {X 151.996,Y 86.170,Z 56.000,A 180.000,B 0.000,C 180.000} C_DIS
LIN {X 152.167,Y 84.561,Z 56.000,A 180.000,B 0.000,C 180.000} C_DIS
LIN {X 152.182,Y 84.383,Z 56.000,A 180.000,B 0.000,C 180.000} C_DIS
LIN {X 152.300,Y 82.952,Z 56.000,A 180.000,B 0.000,C 180.000} C_DIS
LIN {X 152.314,Y 82.774,Z 56.000,A 180.000,B 0.000,C 180.000} C_DIS
LIN {X 152.315,Y 82.761,Z 56.000,A 180.000,B 0.000,C 180.000} C_DIS
LIN {X 152.325,Y 82.595,Z 56.000,A 180.000,B 0.000,C 180.000} C_DIS
LIN {X 152.409,Y 81.165,Z 56.000,A 180.000,B 0.000,C 180.000} C_DIS
LIN {X 152.419,Y 80.986,Z 56.000,A 180.000,B 0.000,C 180.000} C_DIS
LIN {X 152.475,Y 79.377,Z 56.000,A 180.000,B 0.000,C 180.000} C_DIS
LIN {X 152.480,Y 79.198,Z 56.000,A 180.000,B 0.000,C 180.000} C_DIS
LIN {X 152.499,Y 77.589,Z 56.000,A 180.000,B 0.000,C 180.000} C_DIS
LIN {X 152.499,Y 77.411,Z 56.000,A 180.000,B 0.000,C 180.000} C_DIS
LIN {X 152.480,Y 75.802,Z 56.000,A 180.000,B 0.000,C 180.000} C_DIS
LIN {X 152.475,Y 75.623,Z 56.000,A 180.000,B 0.000,C 180.000} C_DIS
LIN {X 152.419,Y 74.014,Z 56.000,A 180.000,B 0.000,C 180.000} C_DIS
LIN {X 152.409,Y 73.835,Z 56.000,A 180.000,B 0.000,C 180.000} C_DIS
LIN {X 152.325,Y 72.405,Z 56.000,A 180.000,B 0.000,C 180.000} C_DIS
LIN {X 152.315,Y 72.239,Z 56.000,A 180.000,B 0.000,C 180.000} C_DIS
LIN {X 152.314,Y 72.226,Z 56.000,A 180.000,B 0.000,C 180.000} C_DIS
LIN {X 152.300,Y 72.048,Z 56.000,A 180.000,B 0.000,C 180.000} C_DIS
LIN {X 152.182,Y 70.617,Z 56.000,A 180.000,B 0.000,C 180.000} C_DIS
LIN {X 152.167,Y 70.439,Z 56.000,A 180.000,B 0.000,C 180.000} C_DIS
LIN {X 151.996,Y 68.830,Z 56.000,A 180.000,B 0.000,C 180.000} C_DIS
LIN {X 151.975,Y 68.651,Z 56.000,A 180.000,B 0.000,C 180.000} C_DIS
LIN {X 151.767,Y 67.042,Z 56.000,A 180.000,B 0.000,C 180.000} C_DIS
LIN {X 151.741,Y 66.863,Z 56.000,A 180.000,B 0.000,C 180.000} C_DIS
LIN {X 151.521,Y 65.433,Z 56.000,A 180.000,B 0.000,C 180.000} C_DIS
LIN {X 151.494,Y 65.254,Z 56.000,A 180.000,B 0.000,C 180.000} C_DIS
LIN {X 151.462,Y 65.075,Z 56.000,A 180.000,B 0.000,C 180.000} C_DIS
LIN {X 151.208,Y 63.645,Z 56.000,A 180.000,B 0.000,C 180.000} C_DIS
LIN {X 151.175,Y 63.467,Z 56.000,A 180.000,B 0.000,C 180.000} C_DIS
LIN {X 150.850,Y 61.858,Z 56.000,A 180.000,B 0.000,C 180.000} C_DIS
LIN {X 150.811,Y 61.679,Z 56.000,A 180.000,B 0.000,C 180.000} C_DIS
LIN {X 150.487,Y 60.249,Z 56.000,A 180.000,B 0.000,C 180.000} C_DIS
LIN {X 150.447,Y 60.070,Z 56.000,A 180.000,B 0.000,C 180.000} C_DIS
LIN {X 150.402,Y 59.891,Z 56.000,A 180.000,B 0.000,C 180.000} C_DIS
LIN {X 150.042,Y 58.461,Z 56.000,A 180.000,B 0.000,C 180.000} C_DIS
LIN {X 149.995,Y 58.282,Z 56.000,A 180.000,B 0.000,C 180.000} C_DIS
LIN {X 149.600,Y 56.852,Z 56.000,A 180.000,B 0.000,C 180.000} C_DIS
LIN {X 149.550,Y 56.673,Z 56.000,A 180.000,B 0.000,C 180.000} C_DIS
LIN {X 149.497,Y 56.495,Z 56.000,A 180.000,B 0.000,C 180.000} C_DIS
LIN {X 149.065,Y 55.064,Z 56.000,A 180.000,B 0.000,C 180.000} C_DIS
LIN {X 149.008,Y 54.886,Z 56.000,A 180.000,B 0.000,C 180.000} C_DIS
LIN {X 148.540,Y 53.455,Z 56.000,A 180.000,B 0.000,C 180.000} C_DIS
LIN {X 148.480,Y 53.277,Z 56.000,A 180.000,B 0.000,C 180.000} C_DIS
LIN {X 147.974,Y 51.847,Z 56.000,A 180.000,B 0.000,C 180.000} C_DIS
LIN {X 147.911,Y 51.668,Z 56.000,A 180.000,B 0.000,C 180.000} C_DIS
LIN {X 147.846,Y 51.496,Z 56.000,A 180.000,B 0.000,C 180.000} C_DIS
LIN {X 147.299,Y 50.059,Z 56.000,A 180.000,B 0.000,C 180.000} C_DIS
LIN {X 147.227,Y 49.880,Z 56.000,A 180.000,B 0.000,C 180.000} C_DIS
LIN {X 146.645,Y 48.450,Z 56.000,A 180.000,B 0.000,C 180.000} C_DIS
LIN {X 146.595,Y 48.331,Z 56.000,A 180.000,B 0.000,C 180.000} C_DIS
LIN {X 145.947,Y 46.841,Z 56.000,A 180.000,B 0.000,C 180.000} C_DIS
LIN {X 145.880,Y 46.692,Z 56.000,A 180.000,B 0.000,C 180.000} C_DIS
LIN {X 145.203,Y 45.232,Z 56.000,A 180.000,B 0.000,C 180.000} C_DIS
LIN {X 145.164,Y 45.151,Z 56.000,A 180.000,B 0.000,C 180.000} C_DIS
LIN {X 144.449,Y 43.697,Z 56.000,A 180.000,B 0.000,C 180.000} C_DIS
LIN {X 144.413,Y 43.623,Z 56.000,A 180.000,B 0.000,C 180.000} C_DIS
LIN {X 144.320,Y 43.444,Z 56.000,A 180.000,B 0.000,C 180.000} C_DIS
LIN {X 143.668,Y 42.193,Z 56.000,A 180.000,B 0.000,C 180.000} C_DIS
LIN {X 143.574,Y 42.014,Z 56.000,A 180.000,B 0.000,C 180.000} C_DIS
LIN {X 142.785,Y 40.584,Z 56.000,A 180.000,B 0.000,C 180.000} C_DIS
LIN {X 142.683,Y 40.405,Z 56.000,A 180.000,B 0.000,C 180.000} C_DIS
LIN {X 141.947,Y 39.141,Z 56.000,A 180.000,B 0.000,C 180.000} C_DIS
LIN {X 141.849,Y 38.975,Z 56.000,A 180.000,B 0.000,C 180.000} C_DIS
LIN {X 141.768,Y 38.842,Z 56.000,A 180.000,B 0.000,C 180.000} C_DIS
LIN {X 140.971,Y 37.545,Z 56.000,A 180.000,B 0.000,C 180.000} C_DIS
LIN {X 140.874,Y 37.393,Z 56.000,A 180.000,B 0.000,C 180.000} C_DIS
LIN {X 140.047,Y 36.115,Z 56.000,A 180.000,B 0.000,C 180.000} C_DIS
LIN {X 139.980,Y 36.012,Z 56.000,A 180.000,B 0.000,C 180.000} C_DIS
LIN {X 139.928,Y 35.936,Z 56.000,A 180.000,B 0.000,C 180.000} C_DIS
LIN {X 139.076,Y 34.685,Z 56.000,A 180.000,B 0.000,C 180.000} C_DIS
LIN {X 138.953,Y 34.506,Z 56.000,A 180.000,B 0.000,C 180.000} C_DIS
LIN {X 138.014,Y 33.194,Z 56.000,A 180.000,B 0.000,C 180.000} C_DIS
LIN {X 137.927,Y 33.076,Z 56.000,A 180.000,B 0.000,C 180.000} C_DIS
LIN {X 136.941,Y 31.765,Z 56.000,A 180.000,B 0.000,C 180.000} C_DIS
LIN {X 136.848,Y 31.646,Z 56.000,A 180.000,B 0.000,C 180.000} C_DIS
LIN {X 135.861,Y 30.394,Z 56.000,A 180.000,B 0.000,C 180.000} C_DIS
LIN {X 135.714,Y 30.215,Z 56.000,A 180.000,B 0.000,C 180.000} C_DIS
LIN {X 134.796,Y 29.106,Z 56.000,A 180.000,B 0.000,C 180.000} C_DIS
LIN {X 134.677,Y 28.964,Z 56.000,A 180.000,B 0.000,C 180.000} C_DIS
LIN {X 133.590,Y 27.713,Z 56.000,A 180.000,B 0.000,C 180.000} C_DIS
LIN {X 133.544,Y 27.660,Z 56.000,A 180.000,B 0.000,C 180.000} C_DIS
LIN {X 133.430,Y 27.534,Z 56.000,A 180.000,B 0.000,C 180.000} C_DIS
LIN {X 132.453,Y 26.461,Z 56.000,A 180.000,B 0.000,C 180.000} C_DIS
LIN {X 132.293,Y 26.289,Z 56.000,A 180.000,B 0.000,C 180.000} C_DIS
LIN {X 131.220,Y 25.165,Z 56.000,A 180.000,B 0.000,C 180.000} C_DIS
LIN {X 131.090,Y 25.031,Z 56.000,A 180.000,B 0.000,C 180.000} C_DIS
LIN {X 129.969,Y 23.910,Z 56.000,A 180.000,B 0.000,C 180.000} C_DIS
LIN {X 129.835,Y 23.780,Z 56.000,A 180.000,B 0.000,C 180.000} C_DIS
LIN {X 128.711,Y 22.707,Z 56.000,A 180.000,B 0.000,C 180.000} C_DIS
LIN {X 128.539,Y 22.547,Z 56.000,A 180.000,B 0.000,C 180.000} C_DIS
LIN {X 127.466,Y 21.570,Z 56.000,A 180.000,B 0.000,C 180.000} C_DIS
LIN {X 127.340,Y 21.456,Z 56.000,A 180.000,B 0.000,C 180.000} C_DIS
LIN {X 127.287,Y 21.410,Z 56.000,A 180.000,B 0.000,C 180.000} C_DIS
LIN {X 126.036,Y 20.323,Z 56.000,A 180.000,B 0.000,C 180.000} C_DIS
LIN {X 125.894,Y 20.204,Z 56.000,A 180.000,B 0.000,C 180.000} C_DIS
LIN {X 124.785,Y 19.286,Z 56.000,A 180.000,B 0.000,C 180.000} C_DIS
LIN {X 124.606,Y 19.139,Z 56.000,A 180.000,B 0.000,C 180.000} C_DIS
LIN {X 123.354,Y 18.152,Z 56.000,A 180.000,B 0.000,C 180.000} C_DIS
LIN {X 123.235,Y 18.059,Z 56.000,A 180.000,B 0.000,C 180.000} C_DIS
LIN {X 121.924,Y 17.073,Z 56.000,A 180.000,B 0.000,C 180.000} C_DIS
LIN {X 121.806,Y 16.986,Z 56.000,A 180.000,B 0.000,C 180.000} C_DIS
LIN {X 120.494,Y 16.047,Z 56.000,A 180.000,B 0.000,C 180.000} C_DIS
LIN {X 120.315,Y 15.924,Z 56.000,A 180.000,B 0.000,C 180.000} C_DIS
LIN {X 119.064,Y 15.072,Z 56.000,A 180.000,B 0.000,C 180.000} C_DIS
LIN {X 118.988,Y 15.020,Z 56.000,A 180.000,B 0.000,C 180.000} C_DIS
LIN {X 118.885,Y 14.953,Z 56.000,A 180.000,B 0.000,C 180.000} C_DIS
LIN {X 117.607,Y 14.126,Z 56.000,A 180.000,B 0.000,C 180.000} C_DIS
LIN {X 117.455,Y 14.029,Z 56.000,A 180.000,B 0.000,C 180.000} C_DIS
LIN {X 116.158,Y 13.232,Z 56.000,A 180.000,B 0.000,C 180.000} C_DIS
LIN {X 116.025,Y 13.151,Z 56.000,A 180.000,B 0.000,C 180.000} C_DIS
LIN {X 115.859,Y 13.053,Z 56.000,A 180.000,B 0.000,C 180.000} C_DIS
LIN {X 114.595,Y 12.317,Z 56.000,A 180.000,B 0.000,C 180.000} C_DIS
LIN {X 114.416,Y 12.215,Z 56.000,A 180.000,B 0.000,C 180.000} C_DIS
LIN {X 112.986,Y 11.426,Z 56.000,A 180.000,B 0.000,C 180.000} C_DIS
LIN {X 112.807,Y 11.332,Z 56.000,A 180.000,B 0.000,C 180.000} C_DIS
LIN {X 111.556,Y 10.680,Z 56.000,A 180.000,B 0.000,C 180.000} C_DIS
LIN {X 111.377,Y 10.587,Z 56.000,A 180.000,B 0.000,C 180.000} C_DIS
LIN {X 111.303,Y 10.551,Z 56.000,A 180.000,B 0.000,C 180.000} C_DIS
LIN {X 109.849,Y 9.836,Z 56.000,A 180.000,B 0.000,C 180.000} C_DIS
LIN {X 109.768,Y 9.797,Z 56.000,A 180.000,B 0.000,C 180.000} C_DIS
LIN {X 108.308,Y 9.120,Z 56.000,A 180.000,B 0.000,C 180.000} C_DIS
LIN {X 108.159,Y 9.053,Z 56.000,A 180.000,B 0.000,C 180.000} C_DIS
LIN {X 106.669,Y 8.405,Z 56.000,A 180.000,B 0.000,C 180.000} C_DIS
LIN {X 106.550,Y 8.355,Z 56.000,A 180.000,B 0.000,C 180.000} C_DIS
LIN {X 105.120,Y 7.773,Z 56.000,A 180.000,B 0.000,C 180.000} C_DIS
LIN {X 104.941,Y 7.701,Z 56.000,A 180.000,B 0.000,C 180.000} C_DIS
LIN {X 103.504,Y 7.154,Z 56.000,A 180.000,B 0.000,C 180.000} C_DIS
LIN {X 103.332,Y 7.089,Z 56.000,A 180.000,B 0.000,C 180.000} C_DIS
LIN {X 103.153,Y 7.026,Z 56.000,A 180.000,B 0.000,C 180.000} C_DIS
LIN {X 101.723,Y 6.520,Z 56.000,A 180.000,B 0.000,C 180.000} C_DIS
LIN {X 101.545,Y 6.460,Z 56.000,A 180.000,B 0.000,C 180.000} C_DIS
LIN {X 100.114,Y 5.992,Z 56.000,A 180.000,B 0.000,C 180.000} C_DIS
LIN {X 99.936,Y 5.935,Z 56.000,A 180.000,B 0.000,C 180.000} C_DIS
LIN {X 98.505,Y 5.503,Z 56.000,A 180.000,B 0.000,C 180.000} C_DIS
LIN {X 98.327,Y 5.450,Z 56.000,A 180.000,B 0.000,C 180.000} C_DIS
LIN {X 98.148,Y 5.400,Z 56.000,A 180.000,B 0.000,C 180.000} C_DIS
LIN {X 96.718,Y 5.005,Z 56.000,A 180.000,B 0.000,C 180.000} C_DIS
LIN {X 96.539,Y 4.958,Z 56.000,A 180.000,B 0.000,C 180.000} C_DIS
LIN {X 95.109,Y 4.598,Z 56.000,A 180.000,B 0.000,C 180.000} C_DIS
LIN {X 94.930,Y 4.554,Z 56.000,A 180.000,B 0.000,C 180.000} C_DIS
LIN {X 94.751,Y 4.513,Z 56.000,A 180.000,B 0.000,C 180.000} C_DIS
LIN {X 93.321,Y 4.189,Z 56.000,A 180.000,B 0.000,C 180.000} C_DIS
LIN {X 93.142,Y 4.150,Z 56.000,A 180.000,B 0.000,C 180.000} C_DIS
LIN {X 91.533,Y 3.825,Z 56.000,A 180.000,B 0.000,C 180.000} C_DIS
LIN {X 91.355,Y 3.792,Z 56.000,A 180.000,B 0.000,C 180.000} C_DIS
LIN {X 89.925,Y 3.538,Z 56.000,A 180.000,B 0.000,C 180.000} C_DIS
LIN {X 89.746,Y 3.506,Z 56.000,A 180.000,B 0.000,C 180.000} C_DIS
LIN {X 89.567,Y 3.479,Z 56.000,A 180.000,B 0.000,C 180.000} C_DIS
LIN {X 88.137,Y 3.259,Z 56.000,A 180.000,B 0.000,C 180.000} C_DIS
LIN {X 87.958,Y 3.233,Z 56.000,A 180.000,B 0.000,C 180.000} C_DIS
LIN {X 86.349,Y 3.025,Z 56.000,A 180.000,B 0.000,C 180.000} C_DIS
LIN {X 86.170,Y 3.004,Z 56.000,A 180.000,B 0.000,C 180.000} C_DIS
LIN {X 84.561,Y 2.833,Z 56.000,A 180.000,B 0.000,C 180.000} C_DIS
LIN {X 84.383,Y 2.818,Z 56.000,A 180.000,B 0.000,C 180.000} C_DIS
LIN {X 82.952,Y 2.700,Z 56.000,A 180.000,B 0.000,C 180.000} C_DIS
LIN {X 82.774,Y 2.686,Z 56.000,A 180.000,B 0.000,C 180.000} C_DIS
LIN {X 82.761,Y 2.685,Z 56.000,A 180.000,B 0.000,C 180.000} C_DIS
LIN {X 82.595,Y 2.675,Z 56.000,A 180.000,B 0.000,C 180.000} C_DIS
LIN {X 81.165,Y 2.591,Z 56.000,A 180.000,B 0.000,C 180.000} C_DIS
LIN {X 80.986,Y 2.581,Z 56.000,A 180.000,B 0.000,C 180.000} C_DIS
LIN {X 79.377,Y 2.525,Z 56.000,A 180.000,B 0.000,C 180.000} C_DIS
LIN {X 79.198,Y 2.520,Z 56.000,A 180.000,B 0.000,C 180.000} C_DIS
LIN {X 77.589,Y 2.501,Z 56.000,A 180.000,B 0.000,C 180.000} C_DIS
LIN {X 77.411,Y 2.501,Z 56.000,A 180.000,B 0.000,C 180.000} C_DIS
LIN {X 75.802,Y 2.520,Z 56.000,A 180.000,B 0.000,C 180.000} C_DIS
LIN {X 75.623,Y 2.525,Z 56.000,A 180.000,B 0.000,C 180.000} C_DIS
LIN {X 74.014,Y 2.581,Z 56.000,A 180.000,B 0.000,C 180.000} C_DIS
LIN {X 73.835,Y 2.591,Z 56.000,A 180.000,B 0.000,C 180.000} C_DIS
LIN {X 72.405,Y 2.675,Z 56.000,A 180.000,B 0.000,C 180.000} C_DIS
LIN {X 72.239,Y 2.685,Z 56.000,A 180.000,B 0.000,C 180.000} C_DIS
LIN {X 72.226,Y 2.686,Z 56.000,A 180.000,B 0.000,C 180.000} C_DIS
LIN {X 72.048,Y 2.700,Z 56.000,A 180.000,B 0.000,C 180.000} C_DIS
LIN {X 70.617,Y 2.818,Z 56.000,A 180.000,B 0.000,C 180.000} C_DIS
LIN {X 70.439,Y 2.833,Z 56.000,A 180.000,B 0.000,C 180.000} C_DIS
LIN {X 68.830,Y 3.004,Z 56.000,A 180.000,B 0.000,C 180.000} C_DIS
LIN {X 68.651,Y 3.025,Z 56.000,A 180.000,B 0.000,C 180.000} C_DIS
LIN {X 67.042,Y 3.233,Z 56.000,A 180.000,B 0.000,C 180.000} C_DIS
LIN {X 66.863,Y 3.259,Z 56.000,A 180.000,B 0.000,C 180.000} C_DIS
LIN {X 65.433,Y 3.479,Z 56.000,A 180.000,B 0.000,C 180.000} C_DIS
LIN {X 65.254,Y 3.506,Z 56.000,A 180.000,B 0.000,C 180.000} C_DIS
LIN {X 65.075,Y 3.538,Z 56.000,A 180.000,B 0.000,C 180.000} C_DIS
LIN {X 63.645,Y 3.792,Z 56.000,A 180.000,B 0.000,C 180.000} C_DIS
LIN {X 63.467,Y 3.825,Z 56.000,A 180.000,B 0.000,C 180.000} C_DIS
LIN {X 61.858,Y 4.150,Z 56.000,A 180.000,B 0.000,C 180.000} C_DIS
LIN {X 61.679,Y 4.189,Z 56.000,A 180.000,B 0.000,C 180.000} C_DIS
LIN {X 60.249,Y 4.513,Z 56.000,A 180.000,B 0.000,C 180.000} C_DIS
LIN {X 60.070,Y 4.554,Z 56.000,A 180.000,B 0.000,C 180.000} C_DIS
LIN {X 59.891,Y 4.598,Z 56.000,A 180.000,B 0.000,C 180.000} C_DIS
LIN {X 58.461,Y 4.958,Z 56.000,A 180.000,B 0.000,C 180.000} C_DIS
LIN {X 58.282,Y 5.005,Z 56.000,A 180.000,B 0.000,C 180.000} C_DIS
LIN {X 56.852,Y 5.400,Z 56.000,A 180.000,B 0.000,C 180.000} C_DIS
LIN {X 56.673,Y 5.450,Z 56.000,A 180.000,B 0.000,C 180.000} C_DIS
LIN {X 56.495,Y 5.503,Z 56.000,A 180.000,B 0.000,C 180.000} C_DIS
LIN {X 55.064,Y 5.935,Z 56.000,A 180.000,B 0.000,C 180.000} C_DIS
LIN {X 54.886,Y 5.992,Z 56.000,A 180.000,B 0.000,C 180.000} C_DIS
LIN {X 53.455,Y 6.460,Z 56.000,A 180.000,B 0.000,C 180.000} C_DIS
LIN {X 53.277,Y 6.520,Z 56.000,A 180.000,B 0.000,C 180.000} C_DIS
LIN {X 51.847,Y 7.026,Z 56.000,A 180.000,B 0.000,C 180.000} C_DIS
LIN {X 51.668,Y 7.089,Z 56.000,A 180.000,B 0.000,C 180.000} C_DIS
LIN {X 51.496,Y 7.154,Z 56.000,A 180.000,B 0.000,C 180.000} C_DIS
LIN {X 50.059,Y 7.701,Z 56.000,A 180.000,B 0.000,C 180.000} C_DIS
LIN {X 49.880,Y 7.773,Z 56.000,A 180.000,B 0.000,C 180.000} C_DIS
LIN {X 48.450,Y 8.355,Z 56.000,A 180.000,B 0.000,C 180.000} C_DIS
LIN {X 48.331,Y 8.405,Z 56.000,A 180.000,B 0.000,C 180.000} C_DIS
LIN {X 46.841,Y 9.053,Z 56.000,A 180.000,B 0.000,C 180.000} C_DIS
LIN {X 46.692,Y 9.120,Z 56.000,A 180.000,B 0.000,C 180.000} C_DIS
LIN {X 45.232,Y 9.797,Z 56.000,A 180.000,B 0.000,C 180.000} C_DIS
LIN {X 45.151,Y 9.836,Z 56.000,A 180.000,B 0.000,C 180.000} C_DIS
LIN {X 43.697,Y 10.551,Z 56.000,A 180.000,B 0.000,C 180.000} C_DIS
LIN {X 43.623,Y 10.587,Z 56.000,A 180.000,B 0.000,C 180.000} C_DIS
LIN {X 43.444,Y 10.680,Z 56.000,A 180.000,B 0.000,C 180.000} C_DIS
LIN {X 42.193,Y 11.332,Z 56.000,A 180.000,B 0.000,C 180.000} C_DIS
LIN {X 42.014,Y 11.426,Z 56.000,A 180.000,B 0.000,C 180.000} C_DIS
LIN {X 40.584,Y 12.215,Z 56.000,A 180.000,B 0.000,C 180.000} C_DIS
LIN {X 40.405,Y 12.317,Z 56.000,A 180.000,B 0.000,C 180.000} C_DIS
LIN {X 39.141,Y 13.053,Z 56.000,A 180.000,B 0.000,C 180.000} C_DIS
LIN {X 38.975,Y 13.151,Z 56.000,A 180.000,B 0.000,C 180.000} C_DIS
LIN {X 38.842,Y 13.232,Z 56.000,A 180.000,B 0.000,C 180.000} C_DIS
LIN {X 37.545,Y 14.029,Z 56.000,A 180.000,B 0.000,C 180.000} C_DIS
LIN {X 37.393,Y 14.126,Z 56.000,A 180.000,B 0.000,C 180.000} C_DIS
LIN {X 36.115,Y 14.953,Z 56.000,A 180.000,B 0.000,C 180.000} C_DIS
LIN {X 36.012,Y 15.020,Z 56.000,A 180.000,B 0.000,C 180.000} C_DIS
LIN {X 35.936,Y 15.072,Z 56.000,A 180.000,B 0.000,C 180.000} C_DIS
LIN {X 34.685,Y 15.924,Z 56.000,A 180.000,B 0.000,C 180.000} C_DIS
LIN {X 34.506,Y 16.047,Z 56.000,A 180.000,B 0.000,C 180.000} C_DIS
LIN {X 33.194,Y 16.986,Z 56.000,A 180.000,B 0.000,C 180.000} C_DIS
LIN {X 33.076,Y 17.073,Z 56.000,A 180.000,B 0.000,C 180.000} C_DIS
LIN {X 31.765,Y 18.059,Z 56.000,A 180.000,B 0.000,C 180.000} C_DIS
LIN {X 31.646,Y 18.152,Z 56.000,A 180.000,B 0.000,C 180.000} C_DIS
LIN {X 30.394,Y 19.139,Z 56.000,A 180.000,B 0.000,C 180.000} C_DIS
LIN {X 30.215,Y 19.286,Z 56.000,A 180.000,B 0.000,C 180.000} C_DIS
LIN {X 29.106,Y 20.204,Z 56.000,A 180.000,B 0.000,C 180.000} C_DIS
LIN {X 28.964,Y 20.323,Z 56.000,A 180.000,B 0.000,C 180.000} C_DIS
LIN {X 27.713,Y 21.410,Z 56.000,A 180.000,B 0.000,C 180.000} C_DIS
LIN {X 27.660,Y 21.456,Z 56.000,A 180.000,B 0.000,C 180.000} C_DIS
LIN {X 27.534,Y 21.570,Z 56.000,A 180.000,B 0.000,C 180.000} C_DIS
LIN {X 26.461,Y 22.547,Z 56.000,A 180.000,B 0.000,C 180.000} C_DIS
LIN {X 26.289,Y 22.707,Z 56.000,A 180.000,B 0.000,C 180.000} C_DIS
LIN {X 25.165,Y 23.780,Z 56.000,A 180.000,B 0.000,C 180.000} C_DIS
LIN {X 25.031,Y 23.910,Z 56.000,A 180.000,B 0.000,C 180.000} C_DIS
LIN {X 23.910,Y 25.031,Z 56.000,A 180.000,B 0.000,C 180.000} C_DIS
LIN {X 23.780,Y 25.165,Z 56.000,A 180.000,B 0.000,C 180.000} C_DIS
LIN {X 22.707,Y 26.289,Z 56.000,A 180.000,B 0.000,C 180.000} C_DIS
LIN {X 22.547,Y 26.461,Z 56.000,A 180.000,B 0.000,C 180.000} C_DIS
LIN {X 21.570,Y 27.534,Z 56.000,A 180.000,B 0.000,C 180.000} C_DIS
LIN {X 21.456,Y 27.660,Z 56.000,A 180.000,B 0.000,C 180.000} C_DIS
LIN {X 21.410,Y 27.713,Z 56.000,A 180.000,B 0.000,C 180.000} C_DIS
LIN {X 20.323,Y 28.964,Z 56.000,A 180.000,B 0.000,C 180.000} C_DIS
LIN {X 20.204,Y 29.106,Z 56.000,A 180.000,B 0.000,C 180.000} C_DIS
LIN {X 19.286,Y 30.215,Z 56.000,A 180.000,B 0.000,C 180.000} C_DIS
LIN {X 19.139,Y 30.394,Z 56.000,A 180.000,B 0.000,C 180.000} C_DIS
LIN {X 18.152,Y 31.646,Z 56.000,A 180.000,B 0.000,C 180.000} C_DIS
LIN {X 18.059,Y 31.765,Z 56.000,A 180.000,B 0.000,C 180.000} C_DIS
LIN {X 17.073,Y 33.076,Z 56.000,A 180.000,B 0.000,C 180.000} C_DIS
LIN {X 16.986,Y 33.194,Z 56.000,A 180.000,B 0.000,C 180.000} C_DIS
LIN {X 16.047,Y 34.506,Z 56.000,A 180.000,B 0.000,C 180.000} C_DIS
LIN {X 15.924,Y 34.685,Z 56.000,A 180.000,B 0.000,C 180.000} C_DIS
LIN {X 15.072,Y 35.936,Z 56.000,A 180.000,B 0.000,C 180.000} C_DIS
LIN {X 15.020,Y 36.012,Z 56.000,A 180.000,B 0.000,C 180.000} C_DIS
LIN {X 14.953,Y 36.115,Z 56.000,A 180.000,B 0.000,C 180.000} C_DIS
LIN {X 14.126,Y 37.393,Z 56.000,A 180.000,B 0.000,C 180.000} C_DIS
LIN {X 14.029,Y 37.545,Z 56.000,A 180.000,B 0.000,C 180.000} C_DIS
LIN {X 13.232,Y 38.842,Z 56.000,A 180.000,B 0.000,C 180.000} C_DIS
LIN {X 13.151,Y 38.975,Z 56.000,A 180.000,B 0.000,C 180.000} C_DIS
LIN {X 13.053,Y 39.141,Z 56.000,A 180.000,B 0.000,C 180.000} C_DIS
LIN {X 12.317,Y 40.405,Z 56.000,A 180.000,B 0.000,C 180.000} C_DIS
LIN {X 12.215,Y 40.584,Z 56.000,A 180.000,B 0.000,C 180.000} C_DIS
LIN {X 11.426,Y 42.014,Z 56.000,A 180.000,B 0.000,C 180.000} C_DIS
LIN {X 11.332,Y 42.193,Z 56.000,A 180.000,B 0.000,C 180.000} C_DIS
LIN {X 10.680,Y 43.444,Z 56.000,A 180.000,B 0.000,C 180.000} C_DIS
LIN {X 10.587,Y 43.623,Z 56.000,A 180.000,B 0.000,C 180.000} C_DIS
LIN {X 10.551,Y 43.697,Z 56.000,A 180.000,B 0.000,C 180.000} C_DIS
LIN {X 9.836,Y 45.151,Z 56.000,A 180.000,B 0.000,C 180.000} C_DIS
LIN {X 9.797,Y 45.232,Z 56.000,A 180.000,B 0.000,C 180.000} C_DIS
LIN {X 9.120,Y 46.692,Z 56.000,A 180.000,B 0.000,C 180.000} C_DIS
LIN {X 9.053,Y 46.841,Z 56.000,A 180.000,B 0.000,C 180.000} C_DIS
LIN {X 8.405,Y 48.331,Z 56.000,A 180.000,B 0.000,C 180.000} C_DIS
LIN {X 8.355,Y 48.450,Z 56.000,A 180.000,B 0.000,C 180.000} C_DIS
LIN {X 7.773,Y 49.880,Z 56.000,A 180.000,B 0.000,C 180.000} C_DIS
LIN {X 7.701,Y 50.059,Z 56.000,A 180.000,B 0.000,C 180.000} C_DIS
LIN {X 7.154,Y 51.496,Z 56.000,A 180.000,B 0.000,C 180.000} C_DIS
LIN {X 7.089,Y 51.668,Z 56.000,A 180.000,B 0.000,C 180.000} C_DIS
LIN {X 7.026,Y 51.847,Z 56.000,A 180.000,B 0.000,C 180.000} C_DIS
LIN {X 6.520,Y 53.277,Z 56.000,A 180.000,B 0.000,C 180.000} C_DIS
LIN {X 6.460,Y 53.455,Z 56.000,A 180.000,B 0.000,C 180.000} C_DIS
LIN {X 5.992,Y 54.886,Z 56.000,A 180.000,B 0.000,C 180.000} C_DIS
LIN {X 5.935,Y 55.064,Z 56.000,A 180.000,B 0.000,C 180.000} C_DIS
LIN {X 5.503,Y 56.495,Z 56.000,A 180.000,B 0.000,C 180.000} C_DIS
LIN {X 5.450,Y 56.673,Z 56.000,A 180.000,B 0.000,C 180.000} C_DIS
LIN {X 5.400,Y 56.852,Z 56.000,A 180.000,B 0.000,C 180.000} C_DIS
LIN {X 5.005,Y 58.282,Z 56.000,A 180.000,B 0.000,C 180.000} C_DIS
LIN {X 4.958,Y 58.461,Z 56.000,A 180.000,B 0.000,C 180.000} C_DIS
LIN {X 4.598,Y 59.891,Z 56.000,A 180.000,B 0.000,C 180.000} C_DIS
LIN {X 4.554,Y 60.070,Z 56.000,A 180.000,B 0.000,C 180.000} C_DIS
LIN {X 4.513,Y 60.249,Z 56.000,A 180.000,B 0.000,C 180.000} C_DIS
LIN {X 4.189,Y 61.679,Z 56.000,A 180.000,B 0.000,C 180.000} C_DIS
LIN {X 4.150,Y 61.858,Z 56.000,A 180.000,B 0.000,C 180.000} C_DIS
LIN {X 3.825,Y 63.467,Z 56.000,A 180.000,B 0.000,C 180.000} C_DIS
LIN {X 3.792,Y 63.645,Z 56.000,A 180.000,B 0.000,C 180.000} C_DIS
LIN {X 3.538,Y 65.075,Z 56.000,A 180.000,B 0.000,C 180.000} C_DIS
LIN {X 3.506,Y 65.254,Z 56.000,A 180.000,B 0.000,C 180.000} C_DIS
LIN {X 3.479,Y 65.433,Z 56.000,A 180.000,B 0.000,C 180.000} C_DIS
LIN {X 3.259,Y 66.863,Z 56.000,A 180.000,B 0.000,C 180.000} C_DIS
LIN {X 3.233,Y 67.042,Z 56.000,A 180.000,B 0.000,C 180.000} C_DIS
LIN {X 3.025,Y 68.651,Z 56.000,A 180.000,B 0.000,C 180.000} C_DIS
LIN {X 3.004,Y 68.830,Z 56.000,A 180.000,B 0.000,C 180.000} C_DIS
LIN {X 2.833,Y 70.439,Z 56.000,A 180.000,B 0.000,C 180.000} C_DIS
LIN {X 2.818,Y 70.617,Z 56.000,A 180.000,B 0.000,C 180.000} C_DIS
LIN {X 2.700,Y 72.048,Z 56.000,A 180.000,B 0.000,C 180.000} C_DIS
LIN {X 2.686,Y 72.226,Z 56.000,A 180.000,B 0.000,C 180.000} C_DIS
LIN {X 2.685,Y 72.239,Z 56.000,A 180.000,B 0.000,C 180.000} C_DIS
LIN {X 2.675,Y 72.405,Z 56.000,A 180.000,B 0.000,C 180.000} C_DIS
LIN {X 2.591,Y 73.835,Z 56.000,A 180.000,B 0.000,C 180.000} C_DIS
LIN {X 2.581,Y 74.014,Z 56.000,A 180.000,B 0.000,C 180.000} C_DIS
LIN {X 2.525,Y 75.623,Z 56.000,A 180.000,B 0.000,C 180.000} C_DIS
LIN {X 2.520,Y 75.802,Z 56.000,A 180.000,B 0.000,C 180.000} C_DIS
LIN {X 2.506,Y 76.973,Z 56.000,A 180.000,B 0.000,C 180.000} C_DIS
LIN {X 2.501,Y 77.411,Z 56.000,A 180.000,B 0.000,C 180.000} C_DIS
LIN {X 2.501,Y 77.589,Z 56.000,A 180.000,B 0.000,C 180.000} C_DIS
LIN {X 2.520,Y 79.198,Z 56.000,A 180.000,B 0.000,C 180.000} C_DIS
LIN {X 2.525,Y 79.377,Z 56.000,A 180.000,B 0.000,C 180.000} C_DIS
LIN {X 2.581,Y 80.986,Z 56.000,A 180.000,B 0.000,C 180.000} C_DIS
LIN {X 2.591,Y 81.165,Z 56.000,A 180.000,B 0.000,C 180.000} C_DIS
LIN {X 2.675,Y 82.595,Z 56.000,A 180.000,B 0.000,C 180.000} C_DIS
LIN {X 2.685,Y 82.761,Z 56.000,A 180.000,B 0.000,C 180.000} C_DIS
LIN {X 2.686,Y 82.774,Z 56.000,A 180.000,B 0.000,C 180.000} C_DIS
LIN {X 2.700,Y 82.952,Z 56.000,A 180.000,B 0.000,C 180.000} C_DIS
LIN {X 2.818,Y 84.383,Z 56.000,A 180.000,B 0.000,C 180.000} C_DIS
LIN {X 2.833,Y 84.561,Z 56.000,A 180.000,B 0.000,C 180.000} C_DIS
LIN {X 3.004,Y 86.170,Z 56.000,A 180.000,B 0.000,C 180.000} C_DIS
LIN {X 3.025,Y 86.349,Z 56.000,A 180.000,B 0.000,C 180.000} C_DIS
LIN {X 3.233,Y 87.958,Z 56.000,A 180.000,B 0.000,C 180.000} C_DIS
LIN {X 3.259,Y 88.137,Z 56.000,A 180.000,B 0.000,C 180.000} C_DIS
LIN {X 3.479,Y 89.567,Z 56.000,A 180.000,B 0.000,C 180.000} C_DIS
LIN {X 3.506,Y 89.746,Z 56.000,A 180.000,B 0.000,C 180.000} C_DIS
LIN {X 3.538,Y 89.925,Z 56.000,A 180.000,B 0.000,C 180.000} C_DIS
LIN {X 3.792,Y 91.355,Z 56.000,A 180.000,B 0.000,C 180.000} C_DIS
LIN {X 3.825,Y 91.533,Z 56.000,A 180.000,B 0.000,C 180.000} C_DIS
LIN {X 4.150,Y 93.142,Z 56.000,A 180.000,B 0.000,C 180.000} C_DIS
LIN {X 4.189,Y 93.321,Z 56.000,A 180.000,B 0.000,C 180.000} C_DIS
LIN {X 4.513,Y 94.751,Z 56.000,A 180.000,B 0.000,C 180.000} C_DIS
LIN {X 4.554,Y 94.930,Z 56.000,A 180.000,B 0.000,C 180.000} C_DIS
LIN {X 4.598,Y 95.109,Z 56.000,A 180.000,B 0.000,C 180.000} C_DIS
LIN {X 4.958,Y 96.539,Z 56.000,A 180.000,B 0.000,C 180.000} C_DIS
LIN {X 5.005,Y 96.718,Z 56.000,A 180.000,B 0.000,C 180.000} C_DIS
LIN {X 5.400,Y 98.148,Z 56.000,A 180.000,B 0.000,C 180.000} C_DIS
LIN {X 5.450,Y 98.327,Z 56.000,A 180.000,B 0.000,C 180.000} C_DIS
LIN {X 5.503,Y 98.505,Z 56.000,A 180.000,B 0.000,C 180.000} C_DIS
LIN {X 5.935,Y 99.936,Z 56.000,A 180.000,B 0.000,C 180.000} C_DIS
LIN {X 5.992,Y 100.114,Z 56.000,A 180.000,B 0.000,C 180.000} C_DIS
LIN {X 6.460,Y 101.545,Z 56.000,A 180.000,B 0.000,C 180.000} C_DIS
LIN {X 6.520,Y 101.723,Z 56.000,A 180.000,B 0.000,C 180.000} C_DIS
LIN {X 7.026,Y 103.153,Z 56.000,A 180.000,B 0.000,C 180.000} C_DIS
LIN {X 7.089,Y 103.332,Z 56.000,A 180.000,B 0.000,C 180.000} C_DIS
LIN {X 7.154,Y 103.504,Z 56.000,A 180.000,B 0.000,C 180.000} C_DIS
LIN {X 7.701,Y 104.941,Z 56.000,A 180.000,B 0.000,C 180.000} C_DIS
LIN {X 7.773,Y 105.120,Z 56.000,A 180.000,B 0.000,C 180.000} C_DIS
LIN {X 8.355,Y 106.550,Z 56.000,A 180.000,B 0.000,C 180.000} C_DIS
LIN {X 8.405,Y 106.669,Z 56.000,A 180.000,B 0.000,C 180.000} C_DIS
